(* CODESYS project 18_CS3_EtherCatIOL
   Company: WAGO Contact SA
   Version: 0.0.0.1

Project tree, tasks and I/O mapping:
  Device : 750-8302 PFC300, WAGO, order no. 750-8302, version 6.4.5.11
    application Application
      libraries: Standard, 3.5.18.0 (System)
      task EtherCAT_Task (cyclic, interval t#4ms, priority 1) calls nothing
      task MainTask (cyclic, interval t#50ms, priority 15) calls PLC_PRG
      global variables GVL_IO
      program PLC_PRG [ST]
      program PRG_IOL_Call [ST]
    EtherCAT_Master : EtherCAT Master, CODESYS, version 4.10.0.0
        settings: NetworkName = 'br1'; NetworkName = "br1"; SelectNetworkByName = False; SrcAddress1 = 48; SrcAddress2 = 3731374440
      IOFLD_01_765_1202 : 765-1202/ 16DIO FLD EC 24V 2A, WAGO Kontakttechnik GmbH u. Co. KG, order no. 765-1202, version Revision=16#00000001
          settings: EnableExpertSettings = True; Physical Address of the Slave = 1001; StationAlias = 1001; FixedPhysicalAdress = True; DC sync0 cycletime = 4000; DC enable = 0; DC sync0 enable = 0; DC sync0 factor = 'x 1'; DC sync0 shift time = 0; DC sync1 cycletime = 4000; DC sync1 enable = 0; DC sync1 factor = 'x 1'; DC sync1 shift time = 0; Latch 0 control = 0; Latch 1 control = 0; Number of SDO = 38; Digital Logic Port X02 Pin 4: 0=Digital Input NO normally open,  1=Digital Input NC normally closed, 2=Digital Output, 3=Static On.Value = 2; Digital Logic Port X02 Pin 2: 0=Digital Input NO normally open,  1=Digital Input NC normally closed, 2=Digital Output, 3=Static On.Value = 2; Digital Logic Port X04 Pin 4: 0=Digital Input NO normally open,  1=Digital Input NC normally closed, 2=Digital Output, 3=Static On.Value = 2; Digital Logic Port X04 Pin 2: 0=Digital Input NO normally open,  1=Digital Input NC normally closed, 2=Digital Output, 3=Static On.Value = 2; Digital Logic Port X06 Pin 4: 0=Digital Input NO normally open,  1=Digital Input NC normally closed, 2=Digital Output, 3=Static On.Value = 2; Digital Logic Port X06 Pin 2: 0=Digital Input NO normally open,  1=Digital Input NC normally closed, 2=Digital Output, 3=Static On.Value = 2; Digital Logic Port X08 Pin 4: 0=Digital Input NO normally open,  1=Digital Input NC normally closed, 2=Digital Output, 3=Static On.Value = 2; Digital Logic Port X08 Pin 2: 0=Digital Input NO normally open,  1=Digital Input NC normally closed, 2=Digital Output, 3=Static On.Value = 2
          output Application.GVL_IO.xIOFLD_01_X02_P4_Out : BOOL  // Process Data (Pin2 + Pin4).Bit2
          output Application.GVL_IO.xIOFLD_01_X02_P2_Out : BOOL  // Process Data (Pin2 + Pin4).Bit3
          output Application.GVL_IO.xIOFLD_01_X04_P4_Out : BOOL  // Process Data (Pin2 + Pin4).Bit6
          output Application.GVL_IO.xIOFLD_01_X04_P2_Out : BOOL  // Process Data (Pin2 + Pin4).Bit7
          output Application.GVL_IO.xIOFLD_01_X06_P4_Out : BOOL  // Process Data (Pin2 + Pin4).Bit10
          output Application.GVL_IO.xIOFLD_01_X06_P2_Out : BOOL  // Process Data (Pin2 + Pin4).Bit11
          output Application.GVL_IO.xIOFLD_01_X08_P4_Out : BOOL  // Process Data (Pin2 + Pin4).Bit14
          output Application.GVL_IO.xIOFLD_01_X08_P2_Out : BOOL  // Process Data (Pin2 + Pin4).Bit15
          input  Application.GVL_IO.xIOFLD_01_X01_P4_In : BOOL  // Process Data (Pin2 + Pin4).Bit0
          input  Application.GVL_IO.xIOFLD_01_X01_P2_In : BOOL  // Process Data (Pin2 + Pin4).Bit1
          input  Application.GVL_IO.xIOFLD_01_X03_P4_In : BOOL  // Process Data (Pin2 + Pin4).Bit4
          input  Application.GVL_IO.xIOFLD_01_X03_P2_In : BOOL  // Process Data (Pin2 + Pin4).Bit5
          input  Application.GVL_IO.xIOFLD_01_X05_P4_In : BOOL  // Process Data (Pin2 + Pin4).Bit8
          input  Application.GVL_IO.xIOFLD_01_X05_P2_In : BOOL  // Process Data (Pin2 + Pin4).Bit9
          input  Application.GVL_IO.xIOFLD_01_X07_P4_In : BOOL  // Process Data (Pin2 + Pin4).Bit12
          input  Application.GVL_IO.xIOFLD_01_X07_P2_In : BOOL  // Process Data (Pin2 + Pin4).Bit13
          unmapped channels: Process Data (Pin2 + Pin4), Control Bit, Toggle Bit, ---, ---, ---, ---, ---, ---, Process Data (Pin2 + Pin4), Status Bit, Toggle Bit, ---, ---, ---, ---, ---, ---, New Message Available Flag, ---, ---, ---, ---, ---, ---, ---
      IOFLD_02_765_4201 : 765-4201/ 8P IOLA FLD EC 24V 2A, WAGO Kontakttechnik GmbH u. Co. KG, order no. 765-4201, version Revision=16#00000001
          settings: ModularDevice = True; MDP_InputOffsets = [0,88,0,152,0,168,184,192,448]; MDP_OutputOffsets = [0,16,80,88,104,112,0,128,0]; Physical Address of the Slave = 1002; StationAlias = 1002; FixedPhysicalAdress = True; Sync.Length = 48; Sync.Length = 57; FMMU.Length = 48; FMMU.Length = 57; Number of RxPDOs of the Slave = 7; Number of TxPDOs of the Slave = 9; DC sync0 cycletime = 4000; DC sync1 cycletime = 4000; Number of SDO = 102; Device ID.Index = 16#8000; Device ID.Subindex = 16#04; Device ID.Value = 0; Device ID.Size = 32; Device ID.AbortIfError = FALSE; Device ID.JumpToLine = FALSE; Device ID.Line = 0; Device ID.CompleteAccess = False; Vendor ID.Index = 16#8000; Vendor ID.Subindex = 16#05; Vendor ID.Value = 0; Vendor ID.Size = 32; Vendor ID.AbortIfError = FALSE; Vendor ID.JumpToLine = FALSE; Vendor ID.Line = 0; Vendor ID.CompleteAccess = False; IO-Link Revision 00 = plausibilty check is deactivate, e.g. 11 = V1.1 - plausibilty check is active.Index = 16#8000; IO-Link Revision 00 = plausibilty check is deactivate, e.g. 11 = V1.1 - plausibilty check is active.Subindex = 16#20; IO-Link Revision 00 = plausibilty check is deactivate, e.g. 11 = V1.1 - plausibilty check is active.Value = 0; IO-Link Revision 00 = plausibilty check is deactivate, e.g. 11 = V1.1 - plausibilty check is active.Size = 8; IO-Link Revision 00 = plausibilty check is deactivate, e.g. 11 = V1.1 - plausibilty check is active.AbortIfError = FALSE; IO-Link Revision 00 = plausibilty check is deactivate, e.g. 11 = V1.1 - plausibilty check is active.JumpToLine = FALSE; IO-Link Revision 00 = plausibilty check is deactivate, e.g. 11 = V1.1 - plausibilty check is active.Line = 0; IO-Link Revision 00 = plausibilty check is deactivate, e.g. 11 = V1.1 - plausibilty check is active.CompleteAccess = False; Cycle Time.Index = 16#8000;
            Cycle Time.Subindex = 16#22; Cycle Time.Value = 0; Cycle Time.Size = 8; Cycle Time.AbortIfError = FALSE; Cycle Time.JumpToLine = FALSE; Cycle Time.Line = 0; Cycle Time.CompleteAccess = False; Configured by the plugged slot module, please do not change..Index = 16#8000; Configured by the plugged slot module, please do not change..Subindex = 16#24; Configured by the plugged slot module, please do not change..Value = 135; Configured by the plugged slot module, please do not change..Size = 8; Configured by the plugged slot module, please do not change..AbortIfError = FALSE; Configured by the plugged slot module, please do not change..JumpToLine = FALSE; Configured by the plugged slot module, please do not change..Line = 0; Configured by the plugged slot module, please do not change..CompleteAccess = False; Configured by the plugged slot module, please do not change..Index = 16#8000; Configured by the plugged slot module, please do not change..Subindex = 16#25; Configured by the plugged slot module, please do not change..Value = 135; Configured by the plugged slot module, please do not change..Size = 8; Configured by the plugged slot module, please do not change..AbortIfError = FALSE; Configured by the plugged slot module, please do not change..JumpToLine = FALSE; Configured by the plugged slot module, please do not change..Line = 0; Configured by the plugged slot module, please do not change..CompleteAccess = False; Master Control: 0x0003 = No Data Storage, 0x0023 = Backup + Restore, 0x0043 = Restore.Index = 16#8000; Master Control: 0x0003 = No Data Storage, 0x0023 = Backup + Restore, 0x0043 = Restore.Subindex = 16#28; Master Control: 0x0003 = No Data Storage, 0x0023 = Backup + Restore, 0x0043 = Restore.Value = 3; Master Control: 0x0003 = No Data Storage, 0x0023 = Backup + Restore, 0x0043 = Restore.Size = 16; Master Control: 0x0003 = No Data Storage, 0x0023 = Backup + Restore, 0x0043 = Restore.AbortIfError = FALSE; Master Control: 0x0003 = No Data Storage, 0x0023 = Backup + Restore, 0x0043 = Restore.JumpToLine = FALSE; Master Control: 0x0003 = No Data Storage, 0x0023 = Backup + Restore, 0x0043 = Restore.Line = 0; Master Control: 0x0003 = No Data Storage, 0x0023 = Backup + Restore, 0x0043 = Restore.CompleteAccess = False; Configured by the plugged slot module, please do not change..Index = 16#2100; Configured by the plugged slot module, please do not change..Subindex = 16#24; Configured by the plugged slot module, please do not change..Value = 8; Configured by the plugged slot module, please do not change..Size = 8; Configured by the plugged slot module, please do not change..AbortIfError = FALSE; Configured by the plugged slot module, please do not change..JumpToLine = FALSE; Configured by the plugged slot module, please do not change..Line = 0; Configured by the plugged slot module, please do not change..CompleteAccess = False; Configured by the plugged slot module, please do not change..Index = 16#2100;
            Configured by the plugged slot module, please do not change..Subindex = 16#25; Configured by the plugged slot module, please do not change..Value = 8; Configured by the plugged slot module, please do not change..Size = 8; Configured by the plugged slot module, please do not change..AbortIfError = FALSE; Configured by the plugged slot module, please do not change..JumpToLine = FALSE; Configured by the plugged slot module, please do not change..Line = 0; Configured by the plugged slot module, please do not change..CompleteAccess = False; Configured by the plugged slot module, please do not change..Index = 16#8010; Configured by the plugged slot module, please do not change..Subindex = 16#24; Configured by the plugged slot module, please do not change..Value = 0; Configured by the plugged slot module, please do not change..Size = 8; Configured by the plugged slot module, please do not change..AbortIfError = FALSE; Configured by the plugged slot module, please do not change..JumpToLine = FALSE; Configured by the plugged slot module, please do not change..Line = 0; Configured by the plugged slot module, please do not change..CompleteAccess = False; Configured by the plugged slot module, please do not change..Index = 16#8010; Configured by the plugged slot module, please do not change..Subindex = 16#25; Configured by the plugged slot module, please do not change..Value = 128; Configured by the plugged slot module, please do not change..Size = 8; Configured by the plugged slot module, please do not change..AbortIfError = FALSE; Configured by the plugged slot module, please do not change..JumpToLine = FALSE; Configured by the plugged slot module, please do not change..Line = 0; Configured by the plugged slot module, please do not change..CompleteAccess = False; Configured by the plugged slot module, please do not change..Index = 16#8010; Configured by the plugged slot module, please do not change..Subindex = 16#28; Configured by the plugged slot module, please do not change..Value = 2; Configured by the plugged slot module, please do not change..Size = 16; Configured by the plugged slot module, please do not change..AbortIfError = FALSE; Configured by the plugged slot module, please do not change..JumpToLine = FALSE; Configured by the plugged slot module, please do not change..Line = 0; Configured by the plugged slot module, please do not change..CompleteAccess = False; Configured by the plugged slot module, please do not change..Index = 16#2110; Configured by the plugged slot module, please do not change..Subindex = 16#24; Configured by the plugged slot module, please do not change..Value = 0; Configured by the plugged slot module, please do not change..Size = 8; Configured by the plugged slot module, please do not change..AbortIfError = FALSE; Configured by the plugged slot module, please do not change..JumpToLine = FALSE; Configured by the plugged slot module, please do not change..Line = 0; Configured by the plugged slot module, please do not change..CompleteAccess = False; Configured by the plugged slot module, please do not change..Index = 16#2110;
            Configured by the plugged slot module, please do not change..Subindex = 16#25; Configured by the plugged slot module, please do not change..Value = 0; Configured by the plugged slot module, please do not change..Size = 8; Configured by the plugged slot module, please do not change..AbortIfError = FALSE; Configured by the plugged slot module, please do not change..JumpToLine = FALSE; Configured by the plugged slot module, please do not change..Line = 0; Configured by the plugged slot module, please do not change..CompleteAccess = False; Device ID.Index = 16#8020; Device ID.Subindex = 16#04; Device ID.Value = 0; Device ID.Size = 32; Device ID.AbortIfError = FALSE; Device ID.JumpToLine = FALSE; Device ID.Line = 0; Device ID.CompleteAccess = False; Vendor ID.Index = 16#8020; Vendor ID.Subindex = 16#05; Vendor ID.Value = 0; Vendor ID.Size = 32; Vendor ID.AbortIfError = FALSE; Vendor ID.JumpToLine = FALSE; Vendor ID.Line = 0; Vendor ID.CompleteAccess = False; IO-Link Revision 00 = plausibilty check is deactivate, e.g. 11 = V1.1 - plausibilty check is active.Index = 16#8020; IO-Link Revision 00 = plausibilty check is deactivate, e.g. 11 = V1.1 - plausibilty check is active.Subindex = 16#20; IO-Link Revision 00 = plausibilty check is deactivate, e.g. 11 = V1.1 - plausibilty check is active.Value = 0; IO-Link Revision 00 = plausibilty check is deactivate, e.g. 11 = V1.1 - plausibilty check is active.Size = 8; IO-Link Revision 00 = plausibilty check is deactivate, e.g. 11 = V1.1 - plausibilty check is active.AbortIfError = FALSE; IO-Link Revision 00 = plausibilty check is deactivate, e.g. 11 = V1.1 - plausibilty check is active.JumpToLine = FALSE; IO-Link Revision 00 = plausibilty check is deactivate, e.g. 11 = V1.1 - plausibilty check is active.Line = 0; IO-Link Revision 00 = plausibilty check is deactivate, e.g. 11 = V1.1 - plausibilty check is active.CompleteAccess = False; Cycle Time.Index = 16#8020; Cycle Time.Subindex = 16#22; Cycle Time.Value = 0; Cycle Time.Size = 8; Cycle Time.AbortIfError = FALSE; Cycle Time.JumpToLine = FALSE; Cycle Time.Line = 0; Cycle Time.CompleteAccess = False; Configured by the plugged slot module, please do not change..Index = 16#8020;
            Configured by the plugged slot module, please do not change..Subindex = 16#24; Configured by the plugged slot module, please do not change..Value = 129; Configured by the plugged slot module, please do not change..Size = 8; Configured by the plugged slot module, please do not change..AbortIfError = FALSE; Configured by the plugged slot module, please do not change..JumpToLine = FALSE; Configured by the plugged slot module, please do not change..Line = 0; Configured by the plugged slot module, please do not change..CompleteAccess = False; Configured by the plugged slot module, please do not change..Index = 16#8020; Configured by the plugged slot module, please do not change..Subindex = 16#25; Configured by the plugged slot module, please do not change..Value = 129; Configured by the plugged slot module, please do not change..Size = 8; Configured by the plugged slot module, please do not change..AbortIfError = FALSE; Configured by the plugged slot module, please do not change..JumpToLine = FALSE; Configured by the plugged slot module, please do not change..Line = 0; Configured by the plugged slot module, please do not change..CompleteAccess = False; Master Control: 0x0003 = No Data Storage, 0x0023 = Backup + Restore, 0x0043 = Restore.Index = 16#8020; Master Control: 0x0003 = No Data Storage, 0x0023 = Backup + Restore, 0x0043 = Restore.Subindex = 16#28; Master Control: 0x0003 = No Data Storage, 0x0023 = Backup + Restore, 0x0043 = Restore.Value = 3; Master Control: 0x0003 = No Data Storage, 0x0023 = Backup + Restore, 0x0043 = Restore.Size = 16; Master Control: 0x0003 = No Data Storage, 0x0023 = Backup + Restore, 0x0043 = Restore.AbortIfError = FALSE; Master Control: 0x0003 = No Data Storage, 0x0023 = Backup + Restore, 0x0043 = Restore.JumpToLine = FALSE; Master Control: 0x0003 = No Data Storage, 0x0023 = Backup + Restore, 0x0043 = Restore.Line = 0; Master Control: 0x0003 = No Data Storage, 0x0023 = Backup + Restore, 0x0043 = Restore.CompleteAccess = False; Configured by the plugged slot module, please do not change..Index = 16#2120; Configured by the plugged slot module, please do not change..Subindex = 16#24; Configured by the plugged slot module, please do not change..Value = 2; Configured by the plugged slot module, please do not change..Size = 8; Configured by the plugged slot module, please do not change..AbortIfError = FALSE; Configured by the plugged slot module, please do not change..JumpToLine = FALSE; Configured by the plugged slot module, please do not change..Line = 0; Configured by the plugged slot module, please do not change..CompleteAccess = False; Configured by the plugged slot module, please do not change..Index = 16#2120; Configured by the plugged slot module, please do not change..Subindex = 16#25; Configured by the plugged slot module, please do not change..Value = 2; Configured by the plugged slot module, please do not change..Size = 8; Configured by the plugged slot module, please do not change..AbortIfError = FALSE; Configured by the plugged slot module, please do not change..JumpToLine = FALSE; Configured by the plugged slot module, please do not change..Line = 0; Configured by the plugged slot module, please do not change..CompleteAccess = False; Configured by the plugged slot module, please do not change..Index = 16#8030;
            Configured by the plugged slot module, please do not change..Subindex = 16#24; Configured by the plugged slot module, please do not change..Value = 0; Configured by the plugged slot module, please do not change..Size = 8; Configured by the plugged slot module, please do not change..AbortIfError = FALSE; Configured by the plugged slot module, please do not change..JumpToLine = FALSE; Configured by the plugged slot module, please do not change..Line = 0; Configured by the plugged slot module, please do not change..CompleteAccess = False; Configured by the plugged slot module, please do not change..Index = 16#8030; Configured by the plugged slot module, please do not change..Subindex = 16#25; Configured by the plugged slot module, please do not change..Value = 128; Configured by the plugged slot module, please do not change..Size = 8; Configured by the plugged slot module, please do not change..AbortIfError = FALSE; Configured by the plugged slot module, please do not change..JumpToLine = FALSE; Configured by the plugged slot module, please do not change..Line = 0; Configured by the plugged slot module, please do not change..CompleteAccess = False; Configured by the plugged slot module, please do not change..Index = 16#8030; Configured by the plugged slot module, please do not change..Subindex = 16#28; Configured by the plugged slot module, please do not change..Value = 2; Configured by the plugged slot module, please do not change..Size = 16; Configured by the plugged slot module, please do not change..AbortIfError = FALSE; Configured by the plugged slot module, please do not change..JumpToLine = FALSE; Configured by the plugged slot module, please do not change..Line = 0; Configured by the plugged slot module, please do not change..CompleteAccess = False; Configured by the plugged slot module, please do not change..Index = 16#2130; Configured by the plugged slot module, please do not change..Subindex = 16#24; Configured by the plugged slot module, please do not change..Value = 0; Configured by the plugged slot module, please do not change..Size = 8; Configured by the plugged slot module, please do not change..AbortIfError = FALSE; Configured by the plugged slot module, please do not change..JumpToLine = FALSE; Configured by the plugged slot module, please do not change..Line = 0; Configured by the plugged slot module, please do not change..CompleteAccess = False; Configured by the plugged slot module, please do not change..Index = 16#2130; Configured by the plugged slot module, please do not change..Subindex = 16#25; Configured by the plugged slot module, please do not change..Value = 0; Configured by the plugged slot module, please do not change..Size = 8; Configured by the plugged slot module, please do not change..AbortIfError = FALSE; Configured by the plugged slot module, please do not change..JumpToLine = FALSE; Configured by the plugged slot module, please do not change..Line = 0; Configured by the plugged slot module, please do not change..CompleteAccess = False; Device ID.Index = 16#8040;
            Device ID.Subindex = 16#04; Device ID.Value = 0; Device ID.Size = 32; Device ID.AbortIfError = FALSE; Device ID.JumpToLine = FALSE; Device ID.Line = 0; Device ID.CompleteAccess = False; Vendor ID.Index = 16#8040; Vendor ID.Subindex = 16#05; Vendor ID.Value = 0; Vendor ID.Size = 32; Vendor ID.AbortIfError = FALSE; Vendor ID.JumpToLine = FALSE; Vendor ID.Line = 0; Vendor ID.CompleteAccess = False; IO-Link Revision 00 = plausibilty check is deactivate, e.g. 11 = V1.1 - plausibilty check is active.Index = 16#8040; IO-Link Revision 00 = plausibilty check is deactivate, e.g. 11 = V1.1 - plausibilty check is active.Subindex = 16#20; IO-Link Revision 00 = plausibilty check is deactivate, e.g. 11 = V1.1 - plausibilty check is active.Value = 0; IO-Link Revision 00 = plausibilty check is deactivate, e.g. 11 = V1.1 - plausibilty check is active.Size = 8; IO-Link Revision 00 = plausibilty check is deactivate, e.g. 11 = V1.1 - plausibilty check is active.AbortIfError = FALSE; IO-Link Revision 00 = plausibilty check is deactivate, e.g. 11 = V1.1 - plausibilty check is active.JumpToLine = FALSE; IO-Link Revision 00 = plausibilty check is deactivate, e.g. 11 = V1.1 - plausibilty check is active.Line = 0; IO-Link Revision 00 = plausibilty check is deactivate, e.g. 11 = V1.1 - plausibilty check is active.CompleteAccess = False; Cycle Time.Index = 16#8040; Cycle Time.Subindex = 16#22; Cycle Time.Value = 0; Cycle Time.Size = 8; Cycle Time.AbortIfError = FALSE; Cycle Time.JumpToLine = FALSE; Cycle Time.Line = 0; Cycle Time.CompleteAccess = False; Configured by the plugged slot module, please do not change..Index = 16#8040; Configured by the plugged slot module, please do not change..Subindex = 16#24; Configured by the plugged slot module, please do not change..Value = 129; Configured by the plugged slot module, please do not change..Size = 8; Configured by the plugged slot module, please do not change..AbortIfError = FALSE; Configured by the plugged slot module, please do not change..JumpToLine = FALSE; Configured by the plugged slot module, please do not change..Line = 0; Configured by the plugged slot module, please do not change..CompleteAccess = False; Configured by the plugged slot module, please do not change..Index = 16#8040;
            Configured by the plugged slot module, please do not change..Subindex = 16#25; Configured by the plugged slot module, please do not change..Value = 129; Configured by the plugged slot module, please do not change..Size = 8; Configured by the plugged slot module, please do not change..AbortIfError = FALSE; Configured by the plugged slot module, please do not change..JumpToLine = FALSE; Configured by the plugged slot module, please do not change..Line = 0; Configured by the plugged slot module, please do not change..CompleteAccess = False; Master Control: 0x0003 = No Data Storage, 0x0023 = Backup + Restore, 0x0043 = Restore.Index = 16#8040; Master Control: 0x0003 = No Data Storage, 0x0023 = Backup + Restore, 0x0043 = Restore.Subindex = 16#28; Master Control: 0x0003 = No Data Storage, 0x0023 = Backup + Restore, 0x0043 = Restore.Value = 3; Master Control: 0x0003 = No Data Storage, 0x0023 = Backup + Restore, 0x0043 = Restore.Size = 16; Master Control: 0x0003 = No Data Storage, 0x0023 = Backup + Restore, 0x0043 = Restore.AbortIfError = FALSE; Master Control: 0x0003 = No Data Storage, 0x0023 = Backup + Restore, 0x0043 = Restore.JumpToLine = FALSE; Master Control: 0x0003 = No Data Storage, 0x0023 = Backup + Restore, 0x0043 = Restore.Line = 0; Master Control: 0x0003 = No Data Storage, 0x0023 = Backup + Restore, 0x0043 = Restore.CompleteAccess = False; Configured by the plugged slot module, please do not change..Index = 16#2140; Configured by the plugged slot module, please do not change..Subindex = 16#24; Configured by the plugged slot module, please do not change..Value = 2; Configured by the plugged slot module, please do not change..Size = 8; Configured by the plugged slot module, please do not change..AbortIfError = FALSE; Configured by the plugged slot module, please do not change..JumpToLine = FALSE; Configured by the plugged slot module, please do not change..Line = 0; Configured by the plugged slot module, please do not change..CompleteAccess = False; Configured by the plugged slot module, please do not change..Index = 16#2140; Configured by the plugged slot module, please do not change..Subindex = 16#25; Configured by the plugged slot module, please do not change..Value = 2; Configured by the plugged slot module, please do not change..Size = 8; Configured by the plugged slot module, please do not change..AbortIfError = FALSE; Configured by the plugged slot module, please do not change..JumpToLine = FALSE; Configured by the plugged slot module, please do not change..Line = 0; Configured by the plugged slot module, please do not change..CompleteAccess = False; Configured by the plugged slot module, please do not change..Index = 16#8050; Configured by the plugged slot module, please do not change..Subindex = 16#24; Configured by the plugged slot module, please do not change..Value = 128; Configured by the plugged slot module, please do not change..Size = 8; Configured by the plugged slot module, please do not change..AbortIfError = FALSE; Configured by the plugged slot module, please do not change..JumpToLine = FALSE; Configured by the plugged slot module, please do not change..Line = 0; Configured by the plugged slot module, please do not change..CompleteAccess = False; Configured by the plugged slot module, please do not change..Index = 16#8050;
            Configured by the plugged slot module, please do not change..Subindex = 16#25; Configured by the plugged slot module, please do not change..Value = 0; Configured by the plugged slot module, please do not change..Size = 8; Configured by the plugged slot module, please do not change..AbortIfError = FALSE; Configured by the plugged slot module, please do not change..JumpToLine = FALSE; Configured by the plugged slot module, please do not change..Line = 0; Configured by the plugged slot module, please do not change..CompleteAccess = False; Configured by the plugged slot module, please do not change..Index = 16#8050; Configured by the plugged slot module, please do not change..Subindex = 16#28; Configured by the plugged slot module, please do not change..Value = 1; Configured by the plugged slot module, please do not change..Size = 16; Configured by the plugged slot module, please do not change..AbortIfError = FALSE; Configured by the plugged slot module, please do not change..JumpToLine = FALSE; Configured by the plugged slot module, please do not change..Line = 0; Configured by the plugged slot module, please do not change..CompleteAccess = False; Configured by the plugged slot module, please do not change..Index = 16#2150; Configured by the plugged slot module, please do not change..Subindex = 16#24; Configured by the plugged slot module, please do not change..Value = 0; Configured by the plugged slot module, please do not change..Size = 8; Configured by the plugged slot module, please do not change..AbortIfError = FALSE; Configured by the plugged slot module, please do not change..JumpToLine = FALSE; Configured by the plugged slot module, please do not change..Line = 0; Configured by the plugged slot module, please do not change..CompleteAccess = False; Configured by the plugged slot module, please do not change..Index = 16#2150; Configured by the plugged slot module, please do not change..Subindex = 16#25; Configured by the plugged slot module, please do not change..Value = 0; Configured by the plugged slot module, please do not change..Size = 8; Configured by the plugged slot module, please do not change..AbortIfError = FALSE; Configured by the plugged slot module, please do not change..JumpToLine = FALSE; Configured by the plugged slot module, please do not change..Line = 0; Configured by the plugged slot module, please do not change..CompleteAccess = False; Device ID.Index = 16#8060; Device ID.Subindex = 16#04; Device ID.Value = 0; Device ID.Size = 32; Device ID.AbortIfError = FALSE; Device ID.JumpToLine = FALSE; Device ID.Line = 0; Device ID.CompleteAccess = False; Vendor ID.Index = 16#8060;
            Vendor ID.Subindex = 16#05; Vendor ID.Value = 0; Vendor ID.Size = 32; Vendor ID.AbortIfError = FALSE; Vendor ID.JumpToLine = FALSE; Vendor ID.Line = 0; Vendor ID.CompleteAccess = False; IO-Link Revision 00 = plausibilty check is deactivate, e.g. 11 = V1.1 - plausibilty check is active.Index = 16#8060; IO-Link Revision 00 = plausibilty check is deactivate, e.g. 11 = V1.1 - plausibilty check is active.Subindex = 16#20; IO-Link Revision 00 = plausibilty check is deactivate, e.g. 11 = V1.1 - plausibilty check is active.Value = 0; IO-Link Revision 00 = plausibilty check is deactivate, e.g. 11 = V1.1 - plausibilty check is active.Size = 8; IO-Link Revision 00 = plausibilty check is deactivate, e.g. 11 = V1.1 - plausibilty check is active.AbortIfError = FALSE; IO-Link Revision 00 = plausibilty check is deactivate, e.g. 11 = V1.1 - plausibilty check is active.JumpToLine = FALSE; IO-Link Revision 00 = plausibilty check is deactivate, e.g. 11 = V1.1 - plausibilty check is active.Line = 0; IO-Link Revision 00 = plausibilty check is deactivate, e.g. 11 = V1.1 - plausibilty check is active.CompleteAccess = False; Cycle Time.Index = 16#8060; Cycle Time.Subindex = 16#22; Cycle Time.Value = 0; Cycle Time.Size = 8; Cycle Time.AbortIfError = FALSE; Cycle Time.JumpToLine = FALSE; Cycle Time.Line = 0; Cycle Time.CompleteAccess = False; Configured by the plugged slot module, please do not change..Index = 16#8060; Configured by the plugged slot module, please do not change..Subindex = 16#24; Configured by the plugged slot module, please do not change..Value = 159; Configured by the plugged slot module, please do not change..Size = 8; Configured by the plugged slot module, please do not change..AbortIfError = FALSE; Configured by the plugged slot module, please do not change..JumpToLine = FALSE; Configured by the plugged slot module, please do not change..Line = 0; Configured by the plugged slot module, please do not change..CompleteAccess = False; Configured by the plugged slot module, please do not change..Index = 16#8060; Configured by the plugged slot module, please do not change..Subindex = 16#25; Configured by the plugged slot module, please do not change..Value = 159; Configured by the plugged slot module, please do not change..Size = 8; Configured by the plugged slot module, please do not change..AbortIfError = FALSE; Configured by the plugged slot module, please do not change..JumpToLine = FALSE; Configured by the plugged slot module, please do not change..Line = 0; Configured by the plugged slot module, please do not change..CompleteAccess = False; Master Control: 0x0003 = No Data Storage, 0x0023 = Backup + Restore, 0x0043 = Restore.Index = 16#8060;
            Master Control: 0x0003 = No Data Storage, 0x0023 = Backup + Restore, 0x0043 = Restore.Subindex = 16#28; Master Control: 0x0003 = No Data Storage, 0x0023 = Backup + Restore, 0x0043 = Restore.Value = 3; Master Control: 0x0003 = No Data Storage, 0x0023 = Backup + Restore, 0x0043 = Restore.Size = 16; Master Control: 0x0003 = No Data Storage, 0x0023 = Backup + Restore, 0x0043 = Restore.AbortIfError = FALSE; Master Control: 0x0003 = No Data Storage, 0x0023 = Backup + Restore, 0x0043 = Restore.JumpToLine = FALSE; Master Control: 0x0003 = No Data Storage, 0x0023 = Backup + Restore, 0x0043 = Restore.Line = 0; Master Control: 0x0003 = No Data Storage, 0x0023 = Backup + Restore, 0x0043 = Restore.CompleteAccess = False; Configured by the plugged slot module, please do not change..Index = 16#2160; Configured by the plugged slot module, please do not change..Subindex = 16#24; Configured by the plugged slot module, please do not change..Value = 32; Configured by the plugged slot module, please do not change..Size = 8; Configured by the plugged slot module, please do not change..AbortIfError = FALSE; Configured by the plugged slot module, please do not change..JumpToLine = FALSE; Configured by the plugged slot module, please do not change..Line = 0; Configured by the plugged slot module, please do not change..CompleteAccess = False; Configured by the plugged slot module, please do not change..Index = 16#2160; Configured by the plugged slot module, please do not change..Subindex = 16#25; Configured by the plugged slot module, please do not change..Value = 32; Configured by the plugged slot module, please do not change..Size = 8; Configured by the plugged slot module, please do not change..AbortIfError = FALSE; Configured by the plugged slot module, please do not change..JumpToLine = FALSE; Configured by the plugged slot module, please do not change..Line = 0; Configured by the plugged slot module, please do not change..CompleteAccess = False; Configured by the plugged slot module, please do not change..Index = 16#8070; Configured by the plugged slot module, please do not change..Subindex = 16#24; Configured by the plugged slot module, please do not change..Value = 128; Configured by the plugged slot module, please do not change..Size = 8; Configured by the plugged slot module, please do not change..AbortIfError = FALSE; Configured by the plugged slot module, please do not change..JumpToLine = FALSE; Configured by the plugged slot module, please do not change..Line = 0; Configured by the plugged slot module, please do not change..CompleteAccess = False; Configured by the plugged slot module, please do not change..Index = 16#8070; Configured by the plugged slot module, please do not change..Subindex = 16#25; Configured by the plugged slot module, please do not change..Value = 0; Configured by the plugged slot module, please do not change..Size = 8; Configured by the plugged slot module, please do not change..AbortIfError = FALSE; Configured by the plugged slot module, please do not change..JumpToLine = FALSE; Configured by the plugged slot module, please do not change..Line = 0; Configured by the plugged slot module, please do not change..CompleteAccess = False; Configured by the plugged slot module, please do not change..Index = 16#8070;
            Configured by the plugged slot module, please do not change..Subindex = 16#28; Configured by the plugged slot module, please do not change..Value = 1; Configured by the plugged slot module, please do not change..Size = 16; Configured by the plugged slot module, please do not change..AbortIfError = FALSE; Configured by the plugged slot module, please do not change..JumpToLine = FALSE; Configured by the plugged slot module, please do not change..Line = 0; Configured by the plugged slot module, please do not change..CompleteAccess = False; Configured by the plugged slot module, please do not change..Index = 16#2170; Configured by the plugged slot module, please do not change..Subindex = 16#24; Configured by the plugged slot module, please do not change..Value = 0; Configured by the plugged slot module, please do not change..Size = 8; Configured by the plugged slot module, please do not change..AbortIfError = FALSE; Configured by the plugged slot module, please do not change..JumpToLine = FALSE; Configured by the plugged slot module, please do not change..Line = 0; Configured by the plugged slot module, please do not change..CompleteAccess = False; Configured by the plugged slot module, please do not change..Index = 16#2170; Configured by the plugged slot module, please do not change..Subindex = 16#25; Configured by the plugged slot module, please do not change..Value = 0; Configured by the plugged slot module, please do not change..Size = 8; Configured by the plugged slot module, please do not change..AbortIfError = FALSE; Configured by the plugged slot module, please do not change..JumpToLine = FALSE; Configured by the plugged slot module, please do not change..Line = 0; Configured by the plugged slot module, please do not change..CompleteAccess = False; Force Mode Setting: 0=Force mode enable, 1=Force mode disable.Index = 16#2000; Force Mode Setting: 0=Force mode enable, 1=Force mode disable.Subindex = 16#00; Force Mode Setting: 0=Force mode enable, 1=Force mode disable.Value = 0; Force Mode Setting: 0=Force mode enable, 1=Force mode disable.Size = 8; Force Mode Setting: 0=Force mode enable, 1=Force mode disable.AbortIfError = FALSE; Force Mode Setting: 0=Force mode enable, 1=Force mode disable.JumpToLine = FALSE; Force Mode Setting: 0=Force mode enable, 1=Force mode disable.Line = 0; Force Mode Setting: 0=Force mode enable, 1=Force mode disable.CompleteAccess = False; PD-Layout Configuration: 0=Port Based, 1=Pin Based.Index = 16#2001; PD-Layout Configuration: 0=Port Based, 1=Pin Based.Subindex = 16#00; PD-Layout Configuration: 0=Port Based, 1=Pin Based.Value = 0; PD-Layout Configuration: 0=Port Based, 1=Pin Based.Size = 8; PD-Layout Configuration: 0=Port Based, 1=Pin Based.AbortIfError = FALSE; PD-Layout Configuration: 0=Port Based, 1=Pin Based.JumpToLine = FALSE; PD-Layout Configuration: 0=Port Based, 1=Pin Based.Line = 0; PD-Layout Configuration: 0=Port Based, 1=Pin Based.CompleteAccess = False; DO Substitute Mode: 0=Set Low, 1=Substitute Value, 2=Hold last.Index = 16#2002;
            DO Substitute Mode: 0=Set Low, 1=Substitute Value, 2=Hold last.Subindex = 16#01; DO Substitute Mode: 0=Set Low, 1=Substitute Value, 2=Hold last.Value = 0; DO Substitute Mode: 0=Set Low, 1=Substitute Value, 2=Hold last.Size = 8; DO Substitute Mode: 0=Set Low, 1=Substitute Value, 2=Hold last.AbortIfError = FALSE; DO Substitute Mode: 0=Set Low, 1=Substitute Value, 2=Hold last.JumpToLine = FALSE; DO Substitute Mode: 0=Set Low, 1=Substitute Value, 2=Hold last.Line = 0; DO Substitute Mode: 0=Set Low, 1=Substitute Value, 2=Hold last.CompleteAccess = False; DO Substitute Value.Index = 16#2002; DO Substitute Value.Subindex = 16#02; DO Substitute Value.Value = 0; DO Substitute Value.Size = 16; DO Substitute Value.AbortIfError = FALSE; DO Substitute Value.JumpToLine = FALSE; DO Substitute Value.Line = 0; DO Substitute Value.CompleteAccess = False; Disable BT: 0=activation of BT interface is allowed, 1=disable activation of BT interface.Index = 16#2003; Disable BT: 0=activation of BT interface is allowed, 1=disable activation of BT interface.Subindex = 16#01; Disable BT: 0=activation of BT interface is allowed, 1=disable activation of BT interface.Value = 0; Disable BT: 0=activation of BT interface is allowed, 1=disable activation of BT interface.Size = 8; Disable BT: 0=activation of BT interface is allowed, 1=disable activation of BT interface.AbortIfError = FALSE; Disable BT: 0=activation of BT interface is allowed, 1=disable activation of BT interface.JumpToLine = FALSE; Disable BT: 0=activation of BT interface is allowed, 1=disable activation of BT interface.Line = 0; Disable BT: 0=activation of BT interface is allowed, 1=disable activation of BT interface.CompleteAccess = False; BT Timeout: Time out to monitor the BT connection in seconds, input range 6..59s.Index = 16#2003; BT Timeout: Time out to monitor the BT connection in seconds, input range 6..59s.Subindex = 16#02; BT Timeout: Time out to monitor the BT connection in seconds, input range 6..59s.Value = 30; BT Timeout: Time out to monitor the BT connection in seconds, input range 6..59s.Size = 16; BT Timeout: Time out to monitor the BT connection in seconds, input range 6..59s.AbortIfError = FALSE; BT Timeout: Time out to monitor the BT connection in seconds, input range 6..59s.JumpToLine = FALSE; BT Timeout: Time out to monitor the BT connection in seconds, input range 6..59s.Line = 0; BT Timeout: Time out to monitor the BT connection in seconds, input range 6..59s.CompleteAccess = False; Port X01 Pin CQ - DI Invert: false=Digital Input NO normally open,  true=Digital Input NC normally closed.Index = 16#2100; Port X01 Pin CQ - DI Invert: false=Digital Input NO normally open,  true=Digital Input NC normally closed.Subindex = 16#01; Port X01 Pin CQ - DI Invert: false=Digital Input NO normally open,  true=Digital Input NC normally closed.Value = 0; Port X01 Pin CQ - DI Invert: false=Digital Input NO normally open,  true=Digital Input NC normally closed.Size = 8; Port X01 Pin CQ - DI Invert: false=Digital Input NO normally open,  true=Digital Input NC normally closed.AbortIfError = FALSE; Port X01 Pin CQ - DI Invert: false=Digital Input NO normally open,  true=Digital Input NC normally closed.JumpToLine = FALSE; Port X01 Pin CQ - DI Invert: false=Digital Input NO normally open,  true=Digital Input NC normally closed.Line = 0; Port X01 Pin CQ - DI Invert: false=Digital Input NO normally open,  true=Digital Input NC normally closed.CompleteAccess = False; Port X01 Pin CQ - DI Filter Time: 0=no Filter, 30=3ms, 150=15ms, 200=20ms.Index = 16#2100;
            Port X01 Pin CQ - DI Filter Time: 0=no Filter, 30=3ms, 150=15ms, 200=20ms.Subindex = 16#02; Port X01 Pin CQ - DI Filter Time: 0=no Filter, 30=3ms, 150=15ms, 200=20ms.Value = 0; Port X01 Pin CQ - DI Filter Time: 0=no Filter, 30=3ms, 150=15ms, 200=20ms.Size = 8; Port X01 Pin CQ - DI Filter Time: 0=no Filter, 30=3ms, 150=15ms, 200=20ms.AbortIfError = FALSE; Port X01 Pin CQ - DI Filter Time: 0=no Filter, 30=3ms, 150=15ms, 200=20ms.JumpToLine = FALSE; Port X01 Pin CQ - DI Filter Time: 0=no Filter, 30=3ms, 150=15ms, 200=20ms.Line = 0; Port X01 Pin CQ - DI Filter Time: 0=no Filter, 30=3ms, 150=15ms, 200=20ms.CompleteAccess = False; Port X01 Pin CQ - DO Static On: false=off, true=on.Index = 16#2100; Port X01 Pin CQ - DO Static On: false=off, true=on.Subindex = 16#03; Port X01 Pin CQ - DO Static On: false=off, true=on.Value = 0; Port X01 Pin CQ - DO Static On: false=off, true=on.Size = 8; Port X01 Pin CQ - DO Static On: false=off, true=on.AbortIfError = FALSE; Port X01 Pin CQ - DO Static On: false=off, true=on.JumpToLine = FALSE; Port X01 Pin CQ - DO Static On: false=off, true=on.Line = 0; Port X01 Pin CQ - DO Static On: false=off, true=on.CompleteAccess = False; Port X01 Pin IQ - Digital Mode: 0=Digital Input NO normally open,  1=Digital Input NC normally closed, 2=Digital Output, 3=Static On, 4=Not supported.Index = 16#2100; Port X01 Pin IQ - Digital Mode: 0=Digital Input NO normally open,  1=Digital Input NC normally closed, 2=Digital Output, 3=Static On, 4=Not supported.Subindex = 16#04; Port X01 Pin IQ - Digital Mode: 0=Digital Input NO normally open,  1=Digital Input NC normally closed, 2=Digital Output, 3=Static On, 4=Not supported.Value = 4; Port X01 Pin IQ - Digital Mode: 0=Digital Input NO normally open,  1=Digital Input NC normally closed, 2=Digital Output, 3=Static On, 4=Not supported.Size = 8; Port X01 Pin IQ - Digital Mode: 0=Digital Input NO normally open,  1=Digital Input NC normally closed, 2=Digital Output, 3=Static On, 4=Not supported.AbortIfError = FALSE; Port X01 Pin IQ - Digital Mode: 0=Digital Input NO normally open,  1=Digital Input NC normally closed, 2=Digital Output, 3=Static On, 4=Not supported.JumpToLine = FALSE; Port X01 Pin IQ - Digital Mode: 0=Digital Input NO normally open,  1=Digital Input NC normally closed, 2=Digital Output, 3=Static On, 4=Not supported.Line = 0; Port X01 Pin IQ - Digital Mode: 0=Digital Input NO normally open,  1=Digital Input NC normally closed, 2=Digital Output, 3=Static On, 4=Not supported.CompleteAccess = False; Port X01 Pin IQ - DI Filter Time: 0=no Filter, 30=3ms, 150=15ms, 200=20ms.Index = 16#2100; Port X01 Pin IQ - DI Filter Time: 0=no Filter, 30=3ms, 150=15ms, 200=20ms.Subindex = 16#05; Port X01 Pin IQ - DI Filter Time: 0=no Filter, 30=3ms, 150=15ms, 200=20ms.Value = 0; Port X01 Pin IQ - DI Filter Time: 0=no Filter, 30=3ms, 150=15ms, 200=20ms.Size = 8; Port X01 Pin IQ - DI Filter Time: 0=no Filter, 30=3ms, 150=15ms, 200=20ms.AbortIfError = FALSE; Port X01 Pin IQ - DI Filter Time: 0=no Filter, 30=3ms, 150=15ms, 200=20ms.JumpToLine = FALSE; Port X01 Pin IQ - DI Filter Time: 0=no Filter, 30=3ms, 150=15ms, 200=20ms.Line = 0; Port X01 Pin IQ - DI Filter Time: 0=no Filter, 30=3ms, 150=15ms, 200=20ms.CompleteAccess = False; Port X02 Pin CQ - DI Invert: false=Digital Input NO normally open,  true=Digital Input NC normally closed.Index = 16#2110; Port X02 Pin CQ - DI Invert: false=Digital Input NO normally open,  true=Digital Input NC normally closed.Subindex = 16#01; Port X02 Pin CQ - DI Invert: false=Digital Input NO normally open,  true=Digital Input NC normally closed.Value = 0; Port X02 Pin CQ - DI Invert: false=Digital Input NO normally open,  true=Digital Input NC normally closed.Size = 8; Port X02 Pin CQ - DI Invert: false=Digital Input NO normally open,  true=Digital Input NC normally closed.AbortIfError = FALSE; Port X02 Pin CQ - DI Invert: false=Digital Input NO normally open,  true=Digital Input NC normally closed.JumpToLine = FALSE; Port X02 Pin CQ - DI Invert: false=Digital Input NO normally open,  true=Digital Input NC normally closed.Line = 0; Port X02 Pin CQ - DI Invert: false=Digital Input NO normally open,  true=Digital Input NC normally closed.CompleteAccess = False; Port X02 Pin CQ - DI Filter Time: 0=no Filter, 30=3ms, 150=15ms, 200=20ms.Index = 16#2110;
            Port X02 Pin CQ - DI Filter Time: 0=no Filter, 30=3ms, 150=15ms, 200=20ms.Subindex = 16#02; Port X02 Pin CQ - DI Filter Time: 0=no Filter, 30=3ms, 150=15ms, 200=20ms.Value = 0; Port X02 Pin CQ - DI Filter Time: 0=no Filter, 30=3ms, 150=15ms, 200=20ms.Size = 8; Port X02 Pin CQ - DI Filter Time: 0=no Filter, 30=3ms, 150=15ms, 200=20ms.AbortIfError = FALSE; Port X02 Pin CQ - DI Filter Time: 0=no Filter, 30=3ms, 150=15ms, 200=20ms.JumpToLine = FALSE; Port X02 Pin CQ - DI Filter Time: 0=no Filter, 30=3ms, 150=15ms, 200=20ms.Line = 0; Port X02 Pin CQ - DI Filter Time: 0=no Filter, 30=3ms, 150=15ms, 200=20ms.CompleteAccess = False; Port X02 Pin CQ - DO Static On: false=off, true=on.Index = 16#2110; Port X02 Pin CQ - DO Static On: false=off, true=on.Subindex = 16#03; Port X02 Pin CQ - DO Static On: false=off, true=on.Value = 0; Port X02 Pin CQ - DO Static On: false=off, true=on.Size = 8; Port X02 Pin CQ - DO Static On: false=off, true=on.AbortIfError = FALSE; Port X02 Pin CQ - DO Static On: false=off, true=on.JumpToLine = FALSE; Port X02 Pin CQ - DO Static On: false=off, true=on.Line = 0; Port X02 Pin CQ - DO Static On: false=off, true=on.CompleteAccess = False; Port X02 Pin IQ - Digital Mode: 0=Digital Input NO normally open,  1=Digital Input NC normally closed, 2=Digital Output, 3=Static On, 4=Not supported.Index = 16#2110; Port X02 Pin IQ - Digital Mode: 0=Digital Input NO normally open,  1=Digital Input NC normally closed, 2=Digital Output, 3=Static On, 4=Not supported.Subindex = 16#04; Port X02 Pin IQ - Digital Mode: 0=Digital Input NO normally open,  1=Digital Input NC normally closed, 2=Digital Output, 3=Static On, 4=Not supported.Value = 4; Port X02 Pin IQ - Digital Mode: 0=Digital Input NO normally open,  1=Digital Input NC normally closed, 2=Digital Output, 3=Static On, 4=Not supported.Size = 8; Port X02 Pin IQ - Digital Mode: 0=Digital Input NO normally open,  1=Digital Input NC normally closed, 2=Digital Output, 3=Static On, 4=Not supported.AbortIfError = FALSE; Port X02 Pin IQ - Digital Mode: 0=Digital Input NO normally open,  1=Digital Input NC normally closed, 2=Digital Output, 3=Static On, 4=Not supported.JumpToLine = FALSE; Port X02 Pin IQ - Digital Mode: 0=Digital Input NO normally open,  1=Digital Input NC normally closed, 2=Digital Output, 3=Static On, 4=Not supported.Line = 0; Port X02 Pin IQ - Digital Mode: 0=Digital Input NO normally open,  1=Digital Input NC normally closed, 2=Digital Output, 3=Static On, 4=Not supported.CompleteAccess = False; Port X02 Pin IQ - DI Filter Time: 0=no Filter, 30=3ms, 150=15ms, 200=20ms.Index = 16#2110; Port X02 Pin IQ - DI Filter Time: 0=no Filter, 30=3ms, 150=15ms, 200=20ms.Subindex = 16#05; Port X02 Pin IQ - DI Filter Time: 0=no Filter, 30=3ms, 150=15ms, 200=20ms.Value = 0; Port X02 Pin IQ - DI Filter Time: 0=no Filter, 30=3ms, 150=15ms, 200=20ms.Size = 8; Port X02 Pin IQ - DI Filter Time: 0=no Filter, 30=3ms, 150=15ms, 200=20ms.AbortIfError = FALSE; Port X02 Pin IQ - DI Filter Time: 0=no Filter, 30=3ms, 150=15ms, 200=20ms.JumpToLine = FALSE; Port X02 Pin IQ - DI Filter Time: 0=no Filter, 30=3ms, 150=15ms, 200=20ms.Line = 0; Port X02 Pin IQ - DI Filter Time: 0=no Filter, 30=3ms, 150=15ms, 200=20ms.CompleteAccess = False; Port X03 Pin CQ - DI Invert: false=Digital Input NO normally open,  true=Digital Input NC normally closed.Index = 16#2120; Port X03 Pin CQ - DI Invert: false=Digital Input NO normally open,  true=Digital Input NC normally closed.Subindex = 16#01; Port X03 Pin CQ - DI Invert: false=Digital Input NO normally open,  true=Digital Input NC normally closed.Value = 0; Port X03 Pin CQ - DI Invert: false=Digital Input NO normally open,  true=Digital Input NC normally closed.Size = 8; Port X03 Pin CQ - DI Invert: false=Digital Input NO normally open,  true=Digital Input NC normally closed.AbortIfError = FALSE; Port X03 Pin CQ - DI Invert: false=Digital Input NO normally open,  true=Digital Input NC normally closed.JumpToLine = FALSE; Port X03 Pin CQ - DI Invert: false=Digital Input NO normally open,  true=Digital Input NC normally closed.Line = 0; Port X03 Pin CQ - DI Invert: false=Digital Input NO normally open,  true=Digital Input NC normally closed.CompleteAccess = False; Port X03 Pin CQ - DI Filter Time: 0=no Filter, 30=3ms, 150=15ms, 200=20ms.Index = 16#2120;
            Port X03 Pin CQ - DI Filter Time: 0=no Filter, 30=3ms, 150=15ms, 200=20ms.Subindex = 16#02; Port X03 Pin CQ - DI Filter Time: 0=no Filter, 30=3ms, 150=15ms, 200=20ms.Value = 0; Port X03 Pin CQ - DI Filter Time: 0=no Filter, 30=3ms, 150=15ms, 200=20ms.Size = 8; Port X03 Pin CQ - DI Filter Time: 0=no Filter, 30=3ms, 150=15ms, 200=20ms.AbortIfError = FALSE; Port X03 Pin CQ - DI Filter Time: 0=no Filter, 30=3ms, 150=15ms, 200=20ms.JumpToLine = FALSE; Port X03 Pin CQ - DI Filter Time: 0=no Filter, 30=3ms, 150=15ms, 200=20ms.Line = 0; Port X03 Pin CQ - DI Filter Time: 0=no Filter, 30=3ms, 150=15ms, 200=20ms.CompleteAccess = False; Port X03 Pin CQ - DO Static On: false=off, true=on.Index = 16#2120; Port X03 Pin CQ - DO Static On: false=off, true=on.Subindex = 16#03; Port X03 Pin CQ - DO Static On: false=off, true=on.Value = 0; Port X03 Pin CQ - DO Static On: false=off, true=on.Size = 8; Port X03 Pin CQ - DO Static On: false=off, true=on.AbortIfError = FALSE; Port X03 Pin CQ - DO Static On: false=off, true=on.JumpToLine = FALSE; Port X03 Pin CQ - DO Static On: false=off, true=on.Line = 0; Port X03 Pin CQ - DO Static On: false=off, true=on.CompleteAccess = False; Port X03 Pin IQ - Digital Mode: 0=Digital Input NO normally open,  1=Digital Input NC normally closed, 2=Digital Output, 3=Static On, 4=Not supported.Index = 16#2120; Port X03 Pin IQ - Digital Mode: 0=Digital Input NO normally open,  1=Digital Input NC normally closed, 2=Digital Output, 3=Static On, 4=Not supported.Subindex = 16#04; Port X03 Pin IQ - Digital Mode: 0=Digital Input NO normally open,  1=Digital Input NC normally closed, 2=Digital Output, 3=Static On, 4=Not supported.Value = 4; Port X03 Pin IQ - Digital Mode: 0=Digital Input NO normally open,  1=Digital Input NC normally closed, 2=Digital Output, 3=Static On, 4=Not supported.Size = 8; Port X03 Pin IQ - Digital Mode: 0=Digital Input NO normally open,  1=Digital Input NC normally closed, 2=Digital Output, 3=Static On, 4=Not supported.AbortIfError = FALSE; Port X03 Pin IQ - Digital Mode: 0=Digital Input NO normally open,  1=Digital Input NC normally closed, 2=Digital Output, 3=Static On, 4=Not supported.JumpToLine = FALSE; Port X03 Pin IQ - Digital Mode: 0=Digital Input NO normally open,  1=Digital Input NC normally closed, 2=Digital Output, 3=Static On, 4=Not supported.Line = 0; Port X03 Pin IQ - Digital Mode: 0=Digital Input NO normally open,  1=Digital Input NC normally closed, 2=Digital Output, 3=Static On, 4=Not supported.CompleteAccess = False; Port X03 Pin IQ - DI Filter Time: 0=no Filter, 30=3ms, 150=15ms, 200=20ms.Index = 16#2120; Port X03 Pin IQ - DI Filter Time: 0=no Filter, 30=3ms, 150=15ms, 200=20ms.Subindex = 16#05; Port X03 Pin IQ - DI Filter Time: 0=no Filter, 30=3ms, 150=15ms, 200=20ms.Value = 0; Port X03 Pin IQ - DI Filter Time: 0=no Filter, 30=3ms, 150=15ms, 200=20ms.Size = 8; Port X03 Pin IQ - DI Filter Time: 0=no Filter, 30=3ms, 150=15ms, 200=20ms.AbortIfError = FALSE; Port X03 Pin IQ - DI Filter Time: 0=no Filter, 30=3ms, 150=15ms, 200=20ms.JumpToLine = FALSE; Port X03 Pin IQ - DI Filter Time: 0=no Filter, 30=3ms, 150=15ms, 200=20ms.Line = 0; Port X03 Pin IQ - DI Filter Time: 0=no Filter, 30=3ms, 150=15ms, 200=20ms.CompleteAccess = False; Port X04 Pin CQ - DI Invert: false=Digital Input NO normally open,  true=Digital Input NC normally closed.Index = 16#2130; Port X04 Pin CQ - DI Invert: false=Digital Input NO normally open,  true=Digital Input NC normally closed.Subindex = 16#01; Port X04 Pin CQ - DI Invert: false=Digital Input NO normally open,  true=Digital Input NC normally closed.Value = 0; Port X04 Pin CQ - DI Invert: false=Digital Input NO normally open,  true=Digital Input NC normally closed.Size = 8; Port X04 Pin CQ - DI Invert: false=Digital Input NO normally open,  true=Digital Input NC normally closed.AbortIfError = FALSE; Port X04 Pin CQ - DI Invert: false=Digital Input NO normally open,  true=Digital Input NC normally closed.JumpToLine = FALSE; Port X04 Pin CQ - DI Invert: false=Digital Input NO normally open,  true=Digital Input NC normally closed.Line = 0; Port X04 Pin CQ - DI Invert: false=Digital Input NO normally open,  true=Digital Input NC normally closed.CompleteAccess = False; Port X04 Pin CQ - DI Filter Time: 0=no Filter, 30=3ms, 150=15ms, 200=20ms.Index = 16#2130;
            Port X04 Pin CQ - DI Filter Time: 0=no Filter, 30=3ms, 150=15ms, 200=20ms.Subindex = 16#02; Port X04 Pin CQ - DI Filter Time: 0=no Filter, 30=3ms, 150=15ms, 200=20ms.Value = 0; Port X04 Pin CQ - DI Filter Time: 0=no Filter, 30=3ms, 150=15ms, 200=20ms.Size = 8; Port X04 Pin CQ - DI Filter Time: 0=no Filter, 30=3ms, 150=15ms, 200=20ms.AbortIfError = FALSE; Port X04 Pin CQ - DI Filter Time: 0=no Filter, 30=3ms, 150=15ms, 200=20ms.JumpToLine = FALSE; Port X04 Pin CQ - DI Filter Time: 0=no Filter, 30=3ms, 150=15ms, 200=20ms.Line = 0; Port X04 Pin CQ - DI Filter Time: 0=no Filter, 30=3ms, 150=15ms, 200=20ms.CompleteAccess = False; Port X04 Pin CQ - DO Static On: false=off, true=on.Index = 16#2130; Port X04 Pin CQ - DO Static On: false=off, true=on.Subindex = 16#03; Port X04 Pin CQ - DO Static On: false=off, true=on.Value = 0; Port X04 Pin CQ - DO Static On: false=off, true=on.Size = 8; Port X04 Pin CQ - DO Static On: false=off, true=on.AbortIfError = FALSE; Port X04 Pin CQ - DO Static On: false=off, true=on.JumpToLine = FALSE; Port X04 Pin CQ - DO Static On: false=off, true=on.Line = 0; Port X04 Pin CQ - DO Static On: false=off, true=on.CompleteAccess = False; Port X04 Pin IQ - Digital Mode: 0=Digital Input NO normally open,  1=Digital Input NC normally closed, 2=Digital Output, 3=Static On, 4=Not supported.Index = 16#2130; Port X04 Pin IQ - Digital Mode: 0=Digital Input NO normally open,  1=Digital Input NC normally closed, 2=Digital Output, 3=Static On, 4=Not supported.Subindex = 16#04; Port X04 Pin IQ - Digital Mode: 0=Digital Input NO normally open,  1=Digital Input NC normally closed, 2=Digital Output, 3=Static On, 4=Not supported.Value = 4; Port X04 Pin IQ - Digital Mode: 0=Digital Input NO normally open,  1=Digital Input NC normally closed, 2=Digital Output, 3=Static On, 4=Not supported.Size = 8; Port X04 Pin IQ - Digital Mode: 0=Digital Input NO normally open,  1=Digital Input NC normally closed, 2=Digital Output, 3=Static On, 4=Not supported.AbortIfError = FALSE; Port X04 Pin IQ - Digital Mode: 0=Digital Input NO normally open,  1=Digital Input NC normally closed, 2=Digital Output, 3=Static On, 4=Not supported.JumpToLine = FALSE; Port X04 Pin IQ - Digital Mode: 0=Digital Input NO normally open,  1=Digital Input NC normally closed, 2=Digital Output, 3=Static On, 4=Not supported.Line = 0; Port X04 Pin IQ - Digital Mode: 0=Digital Input NO normally open,  1=Digital Input NC normally closed, 2=Digital Output, 3=Static On, 4=Not supported.CompleteAccess = False; Port X04 Pin IQ - DI Filter Time: 0=no Filter, 30=3ms, 150=15ms, 200=20ms.Index = 16#2130; Port X04 Pin IQ - DI Filter Time: 0=no Filter, 30=3ms, 150=15ms, 200=20ms.Subindex = 16#05; Port X04 Pin IQ - DI Filter Time: 0=no Filter, 30=3ms, 150=15ms, 200=20ms.Value = 0; Port X04 Pin IQ - DI Filter Time: 0=no Filter, 30=3ms, 150=15ms, 200=20ms.Size = 8; Port X04 Pin IQ - DI Filter Time: 0=no Filter, 30=3ms, 150=15ms, 200=20ms.AbortIfError = FALSE; Port X04 Pin IQ - DI Filter Time: 0=no Filter, 30=3ms, 150=15ms, 200=20ms.JumpToLine = FALSE; Port X04 Pin IQ - DI Filter Time: 0=no Filter, 30=3ms, 150=15ms, 200=20ms.Line = 0; Port X04 Pin IQ - DI Filter Time: 0=no Filter, 30=3ms, 150=15ms, 200=20ms.CompleteAccess = False; Port X05 Pin CQ - DI Invert: false=Digital Input NO normally open,  true=Digital Input NC normally closed.Index = 16#2140; Port X05 Pin CQ - DI Invert: false=Digital Input NO normally open,  true=Digital Input NC normally closed.Subindex = 16#01; Port X05 Pin CQ - DI Invert: false=Digital Input NO normally open,  true=Digital Input NC normally closed.Value = 0; Port X05 Pin CQ - DI Invert: false=Digital Input NO normally open,  true=Digital Input NC normally closed.Size = 8; Port X05 Pin CQ - DI Invert: false=Digital Input NO normally open,  true=Digital Input NC normally closed.AbortIfError = FALSE; Port X05 Pin CQ - DI Invert: false=Digital Input NO normally open,  true=Digital Input NC normally closed.JumpToLine = FALSE; Port X05 Pin CQ - DI Invert: false=Digital Input NO normally open,  true=Digital Input NC normally closed.Line = 0; Port X05 Pin CQ - DI Invert: false=Digital Input NO normally open,  true=Digital Input NC normally closed.CompleteAccess = False; Port X05 Pin CQ - DI Filter Time: 0=no Filter, 30=3ms, 150=15ms, 200=20ms.Index = 16#2140;
            Port X05 Pin CQ - DI Filter Time: 0=no Filter, 30=3ms, 150=15ms, 200=20ms.Subindex = 16#02; Port X05 Pin CQ - DI Filter Time: 0=no Filter, 30=3ms, 150=15ms, 200=20ms.Value = 0; Port X05 Pin CQ - DI Filter Time: 0=no Filter, 30=3ms, 150=15ms, 200=20ms.Size = 8; Port X05 Pin CQ - DI Filter Time: 0=no Filter, 30=3ms, 150=15ms, 200=20ms.AbortIfError = FALSE; Port X05 Pin CQ - DI Filter Time: 0=no Filter, 30=3ms, 150=15ms, 200=20ms.JumpToLine = FALSE; Port X05 Pin CQ - DI Filter Time: 0=no Filter, 30=3ms, 150=15ms, 200=20ms.Line = 0; Port X05 Pin CQ - DI Filter Time: 0=no Filter, 30=3ms, 150=15ms, 200=20ms.CompleteAccess = False; Port X05 Pin CQ - DO Static On: false=off, true=on.Index = 16#2140; Port X05 Pin CQ - DO Static On: false=off, true=on.Subindex = 16#03; Port X05 Pin CQ - DO Static On: false=off, true=on.Value = 0; Port X05 Pin CQ - DO Static On: false=off, true=on.Size = 8; Port X05 Pin CQ - DO Static On: false=off, true=on.AbortIfError = FALSE; Port X05 Pin CQ - DO Static On: false=off, true=on.JumpToLine = FALSE; Port X05 Pin CQ - DO Static On: false=off, true=on.Line = 0; Port X05 Pin CQ - DO Static On: false=off, true=on.CompleteAccess = False; Port X05 Pin IQ - Digital Mode: 0=Digital Input NO normally open,  1=Digital Input NC normally closed, 2=Digital Output, 3=Static On, 4=Not supported.Index = 16#2140; Port X05 Pin IQ - Digital Mode: 0=Digital Input NO normally open,  1=Digital Input NC normally closed, 2=Digital Output, 3=Static On, 4=Not supported.Subindex = 16#04; Port X05 Pin IQ - Digital Mode: 0=Digital Input NO normally open,  1=Digital Input NC normally closed, 2=Digital Output, 3=Static On, 4=Not supported.Value = 4; Port X05 Pin IQ - Digital Mode: 0=Digital Input NO normally open,  1=Digital Input NC normally closed, 2=Digital Output, 3=Static On, 4=Not supported.Size = 8; Port X05 Pin IQ - Digital Mode: 0=Digital Input NO normally open,  1=Digital Input NC normally closed, 2=Digital Output, 3=Static On, 4=Not supported.AbortIfError = FALSE; Port X05 Pin IQ - Digital Mode: 0=Digital Input NO normally open,  1=Digital Input NC normally closed, 2=Digital Output, 3=Static On, 4=Not supported.JumpToLine = FALSE; Port X05 Pin IQ - Digital Mode: 0=Digital Input NO normally open,  1=Digital Input NC normally closed, 2=Digital Output, 3=Static On, 4=Not supported.Line = 0; Port X05 Pin IQ - Digital Mode: 0=Digital Input NO normally open,  1=Digital Input NC normally closed, 2=Digital Output, 3=Static On, 4=Not supported.CompleteAccess = False; Port X05 Pin IQ - DI Filter Time: 0=no Filter, 30=3ms, 150=15ms, 200=20ms.Index = 16#2140; Port X05 Pin IQ - DI Filter Time: 0=no Filter, 30=3ms, 150=15ms, 200=20ms.Subindex = 16#05; Port X05 Pin IQ - DI Filter Time: 0=no Filter, 30=3ms, 150=15ms, 200=20ms.Value = 0; Port X05 Pin IQ - DI Filter Time: 0=no Filter, 30=3ms, 150=15ms, 200=20ms.Size = 8; Port X05 Pin IQ - DI Filter Time: 0=no Filter, 30=3ms, 150=15ms, 200=20ms.AbortIfError = FALSE; Port X05 Pin IQ - DI Filter Time: 0=no Filter, 30=3ms, 150=15ms, 200=20ms.JumpToLine = FALSE; Port X05 Pin IQ - DI Filter Time: 0=no Filter, 30=3ms, 150=15ms, 200=20ms.Line = 0; Port X05 Pin IQ - DI Filter Time: 0=no Filter, 30=3ms, 150=15ms, 200=20ms.CompleteAccess = False; Port X06 Pin CQ - DI Invert: false=Digital Input NO normally open,  true=Digital Input NC normally closed.Index = 16#2150; Port X06 Pin CQ - DI Invert: false=Digital Input NO normally open,  true=Digital Input NC normally closed.Subindex = 16#01; Port X06 Pin CQ - DI Invert: false=Digital Input NO normally open,  true=Digital Input NC normally closed.Value = 0; Port X06 Pin CQ - DI Invert: false=Digital Input NO normally open,  true=Digital Input NC normally closed.Size = 8; Port X06 Pin CQ - DI Invert: false=Digital Input NO normally open,  true=Digital Input NC normally closed.AbortIfError = FALSE; Port X06 Pin CQ - DI Invert: false=Digital Input NO normally open,  true=Digital Input NC normally closed.JumpToLine = FALSE; Port X06 Pin CQ - DI Invert: false=Digital Input NO normally open,  true=Digital Input NC normally closed.Line = 0; Port X06 Pin CQ - DI Invert: false=Digital Input NO normally open,  true=Digital Input NC normally closed.CompleteAccess = False; Port X06 Pin CQ - DI Filter Time: 0=no Filter, 30=3ms, 150=15ms, 200=20ms.Index = 16#2150;
            Port X06 Pin CQ - DI Filter Time: 0=no Filter, 30=3ms, 150=15ms, 200=20ms.Subindex = 16#02; Port X06 Pin CQ - DI Filter Time: 0=no Filter, 30=3ms, 150=15ms, 200=20ms.Value = 0; Port X06 Pin CQ - DI Filter Time: 0=no Filter, 30=3ms, 150=15ms, 200=20ms.Size = 8; Port X06 Pin CQ - DI Filter Time: 0=no Filter, 30=3ms, 150=15ms, 200=20ms.AbortIfError = FALSE; Port X06 Pin CQ - DI Filter Time: 0=no Filter, 30=3ms, 150=15ms, 200=20ms.JumpToLine = FALSE; Port X06 Pin CQ - DI Filter Time: 0=no Filter, 30=3ms, 150=15ms, 200=20ms.Line = 0; Port X06 Pin CQ - DI Filter Time: 0=no Filter, 30=3ms, 150=15ms, 200=20ms.CompleteAccess = False; Port X06 Pin CQ - DO Static On: false=off, true=on.Index = 16#2150; Port X06 Pin CQ - DO Static On: false=off, true=on.Subindex = 16#03; Port X06 Pin CQ - DO Static On: false=off, true=on.Value = 0; Port X06 Pin CQ - DO Static On: false=off, true=on.Size = 8; Port X06 Pin CQ - DO Static On: false=off, true=on.AbortIfError = FALSE; Port X06 Pin CQ - DO Static On: false=off, true=on.JumpToLine = FALSE; Port X06 Pin CQ - DO Static On: false=off, true=on.Line = 0; Port X06 Pin CQ - DO Static On: false=off, true=on.CompleteAccess = False; Port X06 Pin IQ - Digital Mode: 0=Digital Input NO normally open,  1=Digital Input NC normally closed, 2=Digital Output, 3=Static On, 4=Not supported.Index = 16#2150; Port X06 Pin IQ - Digital Mode: 0=Digital Input NO normally open,  1=Digital Input NC normally closed, 2=Digital Output, 3=Static On, 4=Not supported.Subindex = 16#04; Port X06 Pin IQ - Digital Mode: 0=Digital Input NO normally open,  1=Digital Input NC normally closed, 2=Digital Output, 3=Static On, 4=Not supported.Value = 4; Port X06 Pin IQ - Digital Mode: 0=Digital Input NO normally open,  1=Digital Input NC normally closed, 2=Digital Output, 3=Static On, 4=Not supported.Size = 8; Port X06 Pin IQ - Digital Mode: 0=Digital Input NO normally open,  1=Digital Input NC normally closed, 2=Digital Output, 3=Static On, 4=Not supported.AbortIfError = FALSE; Port X06 Pin IQ - Digital Mode: 0=Digital Input NO normally open,  1=Digital Input NC normally closed, 2=Digital Output, 3=Static On, 4=Not supported.JumpToLine = FALSE; Port X06 Pin IQ - Digital Mode: 0=Digital Input NO normally open,  1=Digital Input NC normally closed, 2=Digital Output, 3=Static On, 4=Not supported.Line = 0; Port X06 Pin IQ - Digital Mode: 0=Digital Input NO normally open,  1=Digital Input NC normally closed, 2=Digital Output, 3=Static On, 4=Not supported.CompleteAccess = False; Port X06 Pin IQ - DI Filter Time: 0=no Filter, 30=3ms, 150=15ms, 200=20ms.Index = 16#2150; Port X06 Pin IQ - DI Filter Time: 0=no Filter, 30=3ms, 150=15ms, 200=20ms.Subindex = 16#05; Port X06 Pin IQ - DI Filter Time: 0=no Filter, 30=3ms, 150=15ms, 200=20ms.Value = 0; Port X06 Pin IQ - DI Filter Time: 0=no Filter, 30=3ms, 150=15ms, 200=20ms.Size = 8; Port X06 Pin IQ - DI Filter Time: 0=no Filter, 30=3ms, 150=15ms, 200=20ms.AbortIfError = FALSE; Port X06 Pin IQ - DI Filter Time: 0=no Filter, 30=3ms, 150=15ms, 200=20ms.JumpToLine = FALSE; Port X06 Pin IQ - DI Filter Time: 0=no Filter, 30=3ms, 150=15ms, 200=20ms.Line = 0; Port X06 Pin IQ - DI Filter Time: 0=no Filter, 30=3ms, 150=15ms, 200=20ms.CompleteAccess = False; Port X07 Pin CQ - DI Invert: false=Digital Input NO normally open,  true=Digital Input NC normally closed.Index = 16#2160; Port X07 Pin CQ - DI Invert: false=Digital Input NO normally open,  true=Digital Input NC normally closed.Subindex = 16#01; Port X07 Pin CQ - DI Invert: false=Digital Input NO normally open,  true=Digital Input NC normally closed.Value = 0; Port X07 Pin CQ - DI Invert: false=Digital Input NO normally open,  true=Digital Input NC normally closed.Size = 8; Port X07 Pin CQ - DI Invert: false=Digital Input NO normally open,  true=Digital Input NC normally closed.AbortIfError = FALSE; Port X07 Pin CQ - DI Invert: false=Digital Input NO normally open,  true=Digital Input NC normally closed.JumpToLine = FALSE; Port X07 Pin CQ - DI Invert: false=Digital Input NO normally open,  true=Digital Input NC normally closed.Line = 0; Port X07 Pin CQ - DI Invert: false=Digital Input NO normally open,  true=Digital Input NC normally closed.CompleteAccess = False; Port X07 Pin CQ - DI Filter Time: 0=no Filter, 30=3ms, 150=15ms, 200=20ms.Index = 16#2160;
            Port X07 Pin CQ - DI Filter Time: 0=no Filter, 30=3ms, 150=15ms, 200=20ms.Subindex = 16#02; Port X07 Pin CQ - DI Filter Time: 0=no Filter, 30=3ms, 150=15ms, 200=20ms.Value = 0; Port X07 Pin CQ - DI Filter Time: 0=no Filter, 30=3ms, 150=15ms, 200=20ms.Size = 8; Port X07 Pin CQ - DI Filter Time: 0=no Filter, 30=3ms, 150=15ms, 200=20ms.AbortIfError = FALSE; Port X07 Pin CQ - DI Filter Time: 0=no Filter, 30=3ms, 150=15ms, 200=20ms.JumpToLine = FALSE; Port X07 Pin CQ - DI Filter Time: 0=no Filter, 30=3ms, 150=15ms, 200=20ms.Line = 0; Port X07 Pin CQ - DI Filter Time: 0=no Filter, 30=3ms, 150=15ms, 200=20ms.CompleteAccess = False; Port X07 Pin CQ - DO Static On: false=off, true=on.Index = 16#2160; Port X07 Pin CQ - DO Static On: false=off, true=on.Subindex = 16#03; Port X07 Pin CQ - DO Static On: false=off, true=on.Value = 0; Port X07 Pin CQ - DO Static On: false=off, true=on.Size = 8; Port X07 Pin CQ - DO Static On: false=off, true=on.AbortIfError = FALSE; Port X07 Pin CQ - DO Static On: false=off, true=on.JumpToLine = FALSE; Port X07 Pin CQ - DO Static On: false=off, true=on.Line = 0; Port X07 Pin CQ - DO Static On: false=off, true=on.CompleteAccess = False; Port X07 Pin IQ - Digital Mode: 0=Digital Input NO normally open,  1=Digital Input NC normally closed, 2=Digital Output, 3=Static On, 4=Not supported.Index = 16#2160; Port X07 Pin IQ - Digital Mode: 0=Digital Input NO normally open,  1=Digital Input NC normally closed, 2=Digital Output, 3=Static On, 4=Not supported.Subindex = 16#04; Port X07 Pin IQ - Digital Mode: 0=Digital Input NO normally open,  1=Digital Input NC normally closed, 2=Digital Output, 3=Static On, 4=Not supported.Value = 4; Port X07 Pin IQ - Digital Mode: 0=Digital Input NO normally open,  1=Digital Input NC normally closed, 2=Digital Output, 3=Static On, 4=Not supported.Size = 8; Port X07 Pin IQ - Digital Mode: 0=Digital Input NO normally open,  1=Digital Input NC normally closed, 2=Digital Output, 3=Static On, 4=Not supported.AbortIfError = FALSE; Port X07 Pin IQ - Digital Mode: 0=Digital Input NO normally open,  1=Digital Input NC normally closed, 2=Digital Output, 3=Static On, 4=Not supported.JumpToLine = FALSE; Port X07 Pin IQ - Digital Mode: 0=Digital Input NO normally open,  1=Digital Input NC normally closed, 2=Digital Output, 3=Static On, 4=Not supported.Line = 0; Port X07 Pin IQ - Digital Mode: 0=Digital Input NO normally open,  1=Digital Input NC normally closed, 2=Digital Output, 3=Static On, 4=Not supported.CompleteAccess = False; Port X07 Pin IQ - DI Filter Time: 0=no Filter, 30=3ms, 150=15ms, 200=20ms.Index = 16#2160; Port X07 Pin IQ - DI Filter Time: 0=no Filter, 30=3ms, 150=15ms, 200=20ms.Subindex = 16#05; Port X07 Pin IQ - DI Filter Time: 0=no Filter, 30=3ms, 150=15ms, 200=20ms.Value = 0; Port X07 Pin IQ - DI Filter Time: 0=no Filter, 30=3ms, 150=15ms, 200=20ms.Size = 8; Port X07 Pin IQ - DI Filter Time: 0=no Filter, 30=3ms, 150=15ms, 200=20ms.AbortIfError = FALSE; Port X07 Pin IQ - DI Filter Time: 0=no Filter, 30=3ms, 150=15ms, 200=20ms.JumpToLine = FALSE; Port X07 Pin IQ - DI Filter Time: 0=no Filter, 30=3ms, 150=15ms, 200=20ms.Line = 0; Port X07 Pin IQ - DI Filter Time: 0=no Filter, 30=3ms, 150=15ms, 200=20ms.CompleteAccess = False; Port X08 Pin CQ - DI Invert: false=Digital Input NO normally open,  true=Digital Input NC normally closed.Index = 16#2170; Port X08 Pin CQ - DI Invert: false=Digital Input NO normally open,  true=Digital Input NC normally closed.Subindex = 16#01; Port X08 Pin CQ - DI Invert: false=Digital Input NO normally open,  true=Digital Input NC normally closed.Value = 0; Port X08 Pin CQ - DI Invert: false=Digital Input NO normally open,  true=Digital Input NC normally closed.Size = 8; Port X08 Pin CQ - DI Invert: false=Digital Input NO normally open,  true=Digital Input NC normally closed.AbortIfError = FALSE; Port X08 Pin CQ - DI Invert: false=Digital Input NO normally open,  true=Digital Input NC normally closed.JumpToLine = FALSE; Port X08 Pin CQ - DI Invert: false=Digital Input NO normally open,  true=Digital Input NC normally closed.Line = 0; Port X08 Pin CQ - DI Invert: false=Digital Input NO normally open,  true=Digital Input NC normally closed.CompleteAccess = False; Port X08 Pin CQ - DI Filter Time: 0=no Filter, 30=3ms, 150=15ms, 200=20ms.Index = 16#2170;
            Port X08 Pin CQ - DI Filter Time: 0=no Filter, 30=3ms, 150=15ms, 200=20ms.Subindex = 16#02; Port X08 Pin CQ - DI Filter Time: 0=no Filter, 30=3ms, 150=15ms, 200=20ms.Value = 0; Port X08 Pin CQ - DI Filter Time: 0=no Filter, 30=3ms, 150=15ms, 200=20ms.Size = 8; Port X08 Pin CQ - DI Filter Time: 0=no Filter, 30=3ms, 150=15ms, 200=20ms.AbortIfError = FALSE; Port X08 Pin CQ - DI Filter Time: 0=no Filter, 30=3ms, 150=15ms, 200=20ms.JumpToLine = FALSE; Port X08 Pin CQ - DI Filter Time: 0=no Filter, 30=3ms, 150=15ms, 200=20ms.Line = 0; Port X08 Pin CQ - DI Filter Time: 0=no Filter, 30=3ms, 150=15ms, 200=20ms.CompleteAccess = False; Port X08 Pin CQ - DO Static On: false=off, true=on.Index = 16#2170; Port X08 Pin CQ - DO Static On: false=off, true=on.Subindex = 16#03; Port X08 Pin CQ - DO Static On: false=off, true=on.Value = 0; Port X08 Pin CQ - DO Static On: false=off, true=on.Size = 8; Port X08 Pin CQ - DO Static On: false=off, true=on.AbortIfError = FALSE; Port X08 Pin CQ - DO Static On: false=off, true=on.JumpToLine = FALSE; Port X08 Pin CQ - DO Static On: false=off, true=on.Line = 0; Port X08 Pin CQ - DO Static On: false=off, true=on.CompleteAccess = False; Port X08 Pin IQ - Digital Mode: 0=Digital Input NO normally open,  1=Digital Input NC normally closed, 2=Digital Output, 3=Static On, 4=Not supported.Index = 16#2170; Port X08 Pin IQ - Digital Mode: 0=Digital Input NO normally open,  1=Digital Input NC normally closed, 2=Digital Output, 3=Static On, 4=Not supported.Subindex = 16#04; Port X08 Pin IQ - Digital Mode: 0=Digital Input NO normally open,  1=Digital Input NC normally closed, 2=Digital Output, 3=Static On, 4=Not supported.Value = 4; Port X08 Pin IQ - Digital Mode: 0=Digital Input NO normally open,  1=Digital Input NC normally closed, 2=Digital Output, 3=Static On, 4=Not supported.Size = 8; Port X08 Pin IQ - Digital Mode: 0=Digital Input NO normally open,  1=Digital Input NC normally closed, 2=Digital Output, 3=Static On, 4=Not supported.AbortIfError = FALSE; Port X08 Pin IQ - Digital Mode: 0=Digital Input NO normally open,  1=Digital Input NC normally closed, 2=Digital Output, 3=Static On, 4=Not supported.JumpToLine = FALSE; Port X08 Pin IQ - Digital Mode: 0=Digital Input NO normally open,  1=Digital Input NC normally closed, 2=Digital Output, 3=Static On, 4=Not supported.Line = 0; Port X08 Pin IQ - Digital Mode: 0=Digital Input NO normally open,  1=Digital Input NC normally closed, 2=Digital Output, 3=Static On, 4=Not supported.CompleteAccess = False; Port X08 Pin IQ - DI Filter Time: 0=no Filter, 30=3ms, 150=15ms, 200=20ms.Index = 16#2170; Port X08 Pin IQ - DI Filter Time: 0=no Filter, 30=3ms, 150=15ms, 200=20ms.Subindex = 16#05; Port X08 Pin IQ - DI Filter Time: 0=no Filter, 30=3ms, 150=15ms, 200=20ms.Value = 0; Port X08 Pin IQ - DI Filter Time: 0=no Filter, 30=3ms, 150=15ms, 200=20ms.Size = 8; Port X08 Pin IQ - DI Filter Time: 0=no Filter, 30=3ms, 150=15ms, 200=20ms.AbortIfError = FALSE; Port X08 Pin IQ - DI Filter Time: 0=no Filter, 30=3ms, 150=15ms, 200=20ms.JumpToLine = FALSE; Port X08 Pin IQ - DI Filter Time: 0=no Filter, 30=3ms, 150=15ms, 200=20ms.Line = 0; Port X08 Pin IQ - DI Filter Time: 0=no Filter, 30=3ms, 150=15ms, 200=20ms.CompleteAccess = False; RxTxPdo.NumberofExcludes = 0; RxTxPdo.NumberofEntries = 1; RxTxPdo.Index = 16#1610; RxTxPdo.Fixed = True; RxTxPdo.Mandatory = True; RxTxPdo.Virtual = False; RxTxPdo.Sm = 2; RxTxPdo.Su = 2; RxTxPdo.Name = 'RxPDO Mapping of Digital Outputs';
            RxTxPdo.DependOnSlot = False; RxTxPdo.DependOnSlotGroup = False; RxTxPdo.OverwrittenByModule = False; PD (I/Q Pin2).Index = 16#3001; PD (I/Q Pin2).SubIndex = 1; PD (I/Q Pin2).Size = 16; PD (I/Q Pin2).Offset = 0; PD (I/Q Pin2).DependOnSlot = False; PD (I/Q Pin2).DependOnSlotGroup = False; RxTxPdo.NumberofExcludes = 0; RxTxPdo.NumberofEntries = 8; RxTxPdo.Index = 16#1600; RxTxPdo.Fixed = False; RxTxPdo.Mandatory = False; RxTxPdo.Virtual = False; RxTxPdo.Sm = 2; RxTxPdo.Su = 0; RxTxPdo.Name = 'RxPDO'; RxTxPdo.DependOnSlot = True; RxTxPdo.DependOnSlotGroup = False; RxTxPdo.OverwrittenByModule = True; output byte 0.Index = 16#7000; output byte 0.SubIndex = 1; output byte 0.Size = 8; output byte 0.Offset = 0; output byte 0.DependOnSlot = True; output byte 0.DependOnSlotGroup = False; output byte 1.Index = 16#7000; output byte 1.SubIndex = 2; output byte 1.Size = 8; output byte 1.Offset = 0; output byte 1.DependOnSlot = True; output byte 1.DependOnSlotGroup = False; output byte 2.Index = 16#7000; output byte 2.SubIndex = 3; output byte 2.Size = 8; output byte 2.Offset = 0; output byte 2.DependOnSlot = True; output byte 2.DependOnSlotGroup = False; output byte 3.Index = 16#7000;
            output byte 3.SubIndex = 4; output byte 3.Size = 8; output byte 3.Offset = 0; output byte 3.DependOnSlot = True; output byte 3.DependOnSlotGroup = False; output byte 4.Index = 16#7000; output byte 4.SubIndex = 5; output byte 4.Size = 8; output byte 4.Offset = 0; output byte 4.DependOnSlot = True; output byte 4.DependOnSlotGroup = False; output byte 5.Index = 16#7000; output byte 5.SubIndex = 6; output byte 5.Size = 8; output byte 5.Offset = 0; output byte 5.DependOnSlot = True; output byte 5.DependOnSlotGroup = False; output byte 6.Index = 16#7000; output byte 6.SubIndex = 7; output byte 6.Size = 8; output byte 6.Offset = 0; output byte 6.DependOnSlot = True; output byte 6.DependOnSlotGroup = False; output byte 7.Index = 16#7000; output byte 7.SubIndex = 8; output byte 7.Size = 8; output byte 7.Offset = 0; output byte 7.DependOnSlot = True; output byte 7.DependOnSlotGroup = False; RxTxPdo.NumberofExcludes = 0; RxTxPdo.NumberofEntries = 1; RxTxPdo.Index = 16#1601; RxTxPdo.Fixed = False; RxTxPdo.Mandatory = False; RxTxPdo.Virtual = False; RxTxPdo.Sm = 2; RxTxPdo.Su = 0; RxTxPdo.Name = 'RxPDO'; RxTxPdo.DependOnSlot = True; RxTxPdo.DependOnSlotGroup = False;
            RxTxPdo.OverwrittenByModule = True; PD (C/Q Pin4).Index = 16#7010; PD (C/Q Pin4).SubIndex = 1; PD (C/Q Pin4).Size = 8; PD (C/Q Pin4).Offset = 0; PD (C/Q Pin4).DependOnSlot = True; PD (C/Q Pin4).DependOnSlotGroup = False; RxTxPdo.NumberofExcludes = 0; RxTxPdo.NumberofEntries = 2; RxTxPdo.Index = 16#1602; RxTxPdo.Fixed = False; RxTxPdo.Mandatory = False; RxTxPdo.Virtual = False; RxTxPdo.Sm = 2; RxTxPdo.Su = 0; RxTxPdo.Name = 'RxPDO'; RxTxPdo.DependOnSlot = True; RxTxPdo.DependOnSlotGroup = False; RxTxPdo.OverwrittenByModule = True; output byte 0.Index = 16#7020; output byte 0.SubIndex = 1; output byte 0.Size = 8; output byte 0.Offset = 0; output byte 0.DependOnSlot = True; output byte 0.DependOnSlotGroup = False; output byte 1.Index = 16#7020; output byte 1.SubIndex = 2; output byte 1.Size = 8; output byte 1.Offset = 0; output byte 1.DependOnSlot = True; output byte 1.DependOnSlotGroup = False; RxTxPdo.NumberofExcludes = 0; RxTxPdo.NumberofEntries = 1; RxTxPdo.Index = 16#1603; RxTxPdo.Fixed = False; RxTxPdo.Mandatory = False; RxTxPdo.Virtual = False; RxTxPdo.Sm = 2; RxTxPdo.Su = 0; RxTxPdo.Name = 'RxPDO';
            RxTxPdo.DependOnSlot = True; RxTxPdo.DependOnSlotGroup = False; RxTxPdo.OverwrittenByModule = True; PD (C/Q Pin4).Index = 16#7030; PD (C/Q Pin4).SubIndex = 1; PD (C/Q Pin4).Size = 8; PD (C/Q Pin4).Offset = 0; PD (C/Q Pin4).DependOnSlot = True; PD (C/Q Pin4).DependOnSlotGroup = False; RxTxPdo.NumberofExcludes = 0; RxTxPdo.NumberofEntries = 2; RxTxPdo.Index = 16#1604; RxTxPdo.Fixed = False; RxTxPdo.Mandatory = False; RxTxPdo.Virtual = False; RxTxPdo.Sm = 2; RxTxPdo.Su = 0; RxTxPdo.Name = 'RxPDO'; RxTxPdo.DependOnSlot = True; RxTxPdo.DependOnSlotGroup = False; RxTxPdo.OverwrittenByModule = True; output byte 0.Index = 16#7040; output byte 0.SubIndex = 1; output byte 0.Size = 8; output byte 0.Offset = 0; output byte 0.DependOnSlot = True; output byte 0.DependOnSlotGroup = False; output byte 1.Index = 16#7040; output byte 1.SubIndex = 2; output byte 1.Size = 8; output byte 1.Offset = 0; output byte 1.DependOnSlot = True; output byte 1.DependOnSlotGroup = False; RxTxPdo.NumberofExcludes = 0; RxTxPdo.NumberofEntries = 32; RxTxPdo.Index = 16#1606; RxTxPdo.Fixed = False; RxTxPdo.Mandatory = False; RxTxPdo.Virtual = False; RxTxPdo.Sm = 2;
            RxTxPdo.Su = 0; RxTxPdo.Name = 'RxPDO'; RxTxPdo.DependOnSlot = True; RxTxPdo.DependOnSlotGroup = False; RxTxPdo.OverwrittenByModule = True; output byte 0.Index = 16#7060; output byte 0.SubIndex = 1; output byte 0.Size = 8; output byte 0.Offset = 0; output byte 0.DependOnSlot = True; output byte 0.DependOnSlotGroup = False; output byte 1.Index = 16#7060; output byte 1.SubIndex = 2; output byte 1.Size = 8; output byte 1.Offset = 0; output byte 1.DependOnSlot = True; output byte 1.DependOnSlotGroup = False; output byte 2.Index = 16#7060; output byte 2.SubIndex = 3; output byte 2.Size = 8; output byte 2.Offset = 0; output byte 2.DependOnSlot = True; output byte 2.DependOnSlotGroup = False; output byte 3.Index = 16#7060; output byte 3.SubIndex = 4; output byte 3.Size = 8; output byte 3.Offset = 0; output byte 3.DependOnSlot = True; output byte 3.DependOnSlotGroup = False; output byte 4.Index = 16#7060; output byte 4.SubIndex = 5; output byte 4.Size = 8; output byte 4.Offset = 0; output byte 4.DependOnSlot = True; output byte 4.DependOnSlotGroup = False; output byte 5.Index = 16#7060; output byte 5.SubIndex = 6; output byte 5.Size = 8; output byte 5.Offset = 0; output byte 5.DependOnSlot = True;
            output byte 5.DependOnSlotGroup = False; output byte 6.Index = 16#7060; output byte 6.SubIndex = 7; output byte 6.Size = 8; output byte 6.Offset = 0; output byte 6.DependOnSlot = True; output byte 6.DependOnSlotGroup = False; output byte 7.Index = 16#7060; output byte 7.SubIndex = 8; output byte 7.Size = 8; output byte 7.Offset = 0; output byte 7.DependOnSlot = True; output byte 7.DependOnSlotGroup = False; output byte 8.Index = 16#7060; output byte 8.SubIndex = 9; output byte 8.Size = 8; output byte 8.Offset = 0; output byte 8.DependOnSlot = True; output byte 8.DependOnSlotGroup = False; output byte 9.Index = 16#7060; output byte 9.SubIndex = 10; output byte 9.Size = 8; output byte 9.Offset = 0; output byte 9.DependOnSlot = True; output byte 9.DependOnSlotGroup = False; output byte 10.Index = 16#7060; output byte 10.SubIndex = 11; output byte 10.Size = 8; output byte 10.Offset = 0; output byte 10.DependOnSlot = True; output byte 10.DependOnSlotGroup = False; output byte 11.Index = 16#7060; output byte 11.SubIndex = 12; output byte 11.Size = 8; output byte 11.Offset = 0; output byte 11.DependOnSlot = True; output byte 11.DependOnSlotGroup = False; output byte 12.Index = 16#7060; output byte 12.SubIndex = 13; output byte 12.Size = 8;
            output byte 12.Offset = 0; output byte 12.DependOnSlot = True; output byte 12.DependOnSlotGroup = False; output byte 13.Index = 16#7060; output byte 13.SubIndex = 14; output byte 13.Size = 8; output byte 13.Offset = 0; output byte 13.DependOnSlot = True; output byte 13.DependOnSlotGroup = False; output byte 14.Index = 16#7060; output byte 14.SubIndex = 15; output byte 14.Size = 8; output byte 14.Offset = 0; output byte 14.DependOnSlot = True; output byte 14.DependOnSlotGroup = False; output byte 15.Index = 16#7060; output byte 15.SubIndex = 16; output byte 15.Size = 8; output byte 15.Offset = 0; output byte 15.DependOnSlot = True; output byte 15.DependOnSlotGroup = False; output byte 16.Index = 16#7060; output byte 16.SubIndex = 17; output byte 16.Size = 8; output byte 16.Offset = 0; output byte 16.DependOnSlot = True; output byte 16.DependOnSlotGroup = False; output byte 17.Index = 16#7060; output byte 17.SubIndex = 18; output byte 17.Size = 8; output byte 17.Offset = 0; output byte 17.DependOnSlot = True; output byte 17.DependOnSlotGroup = False; output byte 18.Index = 16#7060; output byte 18.SubIndex = 19; output byte 18.Size = 8; output byte 18.Offset = 0; output byte 18.DependOnSlot = True; output byte 18.DependOnSlotGroup = False; output byte 19.Index = 16#7060;
            output byte 19.SubIndex = 20; output byte 19.Size = 8; output byte 19.Offset = 0; output byte 19.DependOnSlot = True; output byte 19.DependOnSlotGroup = False; output byte 20.Index = 16#7060; output byte 20.SubIndex = 21; output byte 20.Size = 8; output byte 20.Offset = 0; output byte 20.DependOnSlot = True; output byte 20.DependOnSlotGroup = False; output byte 21.Index = 16#7060; output byte 21.SubIndex = 22; output byte 21.Size = 8; output byte 21.Offset = 0; output byte 21.DependOnSlot = True; output byte 21.DependOnSlotGroup = False; output byte 22.Index = 16#7060; output byte 22.SubIndex = 23; output byte 22.Size = 8; output byte 22.Offset = 0; output byte 22.DependOnSlot = True; output byte 22.DependOnSlotGroup = False; output byte 23.Index = 16#7060; output byte 23.SubIndex = 24; output byte 23.Size = 8; output byte 23.Offset = 0; output byte 23.DependOnSlot = True; output byte 23.DependOnSlotGroup = False; output byte 24.Index = 16#7060; output byte 24.SubIndex = 25; output byte 24.Size = 8; output byte 24.Offset = 0; output byte 24.DependOnSlot = True; output byte 24.DependOnSlotGroup = False; output byte 25.Index = 16#7060; output byte 25.SubIndex = 26; output byte 25.Size = 8; output byte 25.Offset = 0; output byte 25.DependOnSlot = True;
            output byte 25.DependOnSlotGroup = False; output byte 26.Index = 16#7060; output byte 26.SubIndex = 27; output byte 26.Size = 8; output byte 26.Offset = 0; output byte 26.DependOnSlot = True; output byte 26.DependOnSlotGroup = False; output byte 27.Index = 16#7060; output byte 27.SubIndex = 28; output byte 27.Size = 8; output byte 27.Offset = 0; output byte 27.DependOnSlot = True; output byte 27.DependOnSlotGroup = False; output byte 28.Index = 16#7060; output byte 28.SubIndex = 29; output byte 28.Size = 8; output byte 28.Offset = 0; output byte 28.DependOnSlot = True; output byte 28.DependOnSlotGroup = False; output byte 29.Index = 16#7060; output byte 29.SubIndex = 30; output byte 29.Size = 8; output byte 29.Offset = 0; output byte 29.DependOnSlot = True; output byte 29.DependOnSlotGroup = False; output byte 30.Index = 16#7060; output byte 30.SubIndex = 31; output byte 30.Size = 8; output byte 30.Offset = 0; output byte 30.DependOnSlot = True; output byte 30.DependOnSlotGroup = False; output byte 31.Index = 16#7060; output byte 31.SubIndex = 32; output byte 31.Size = 8; output byte 31.Offset = 0; output byte 31.DependOnSlot = True; output byte 31.DependOnSlotGroup = False; RxTxPdo.NumberofExcludes = 0; RxTxPdo.NumberofEntries = 1; RxTxPdo.Index = 16#1A10;
            RxTxPdo.Fixed = True; RxTxPdo.Mandatory = True; RxTxPdo.Virtual = False; RxTxPdo.Sm = 3; RxTxPdo.Su = 3; RxTxPdo.Name = 'TxPDO Mapping of Digital Inputs'; RxTxPdo.DependOnSlot = False; RxTxPdo.DependOnSlotGroup = False; RxTxPdo.OverwrittenByModule = False; PD (I/Q Pin2 + C/Q Pin4).Index = 16#3000; PD (I/Q Pin2 + C/Q Pin4).SubIndex = 1; PD (I/Q Pin2 + C/Q Pin4).Size = 16; PD (I/Q Pin2 + C/Q Pin4).Offset = 0; PD (I/Q Pin2 + C/Q Pin4).DependOnSlot = False; PD (I/Q Pin2 + C/Q Pin4).DependOnSlotGroup = False; RxTxPdo.NumberofExcludes = 0; RxTxPdo.NumberofEntries = 2; RxTxPdo.Index = 16#1A11; RxTxPdo.Fixed = True; RxTxPdo.Mandatory = True; RxTxPdo.Virtual = False; RxTxPdo.Sm = 3; RxTxPdo.Su = 3; RxTxPdo.Name = 'TxPDO Mapping of New Messages Available'; RxTxPdo.DependOnSlot = False; RxTxPdo.DependOnSlotGroup = False; RxTxPdo.OverwrittenByModule = False; New Message Available Flag.Index = 16#10F3; New Message Available Flag.SubIndex = 4; New Message Available Flag.Size = 1; New Message Available Flag.Offset = 0; New Message Available Flag.DependOnSlot = False; New Message Available Flag.DependOnSlotGroup = False; Dummy.Index = 16#0000; Dummy.SubIndex = 0; Dummy.Size = 7; Dummy.Offset = 0; Dummy.DependOnSlot = False; Dummy.DependOnSlotGroup = False; RxTxPdo.NumberofExcludes = 0;
            RxTxPdo.NumberofEntries = 8; RxTxPdo.Index = 16#1A80; RxTxPdo.Fixed = True; RxTxPdo.Mandatory = True; RxTxPdo.Virtual = False; RxTxPdo.Sm = 3; RxTxPdo.Su = 3; RxTxPdo.Name = 'TxPDO Mapping of Status Data'; RxTxPdo.DependOnSlot = False; RxTxPdo.DependOnSlotGroup = False; RxTxPdo.OverwrittenByModule = False; State of IO-Link Port X01.Index = 16#F100; State of IO-Link Port X01.SubIndex = 1; State of IO-Link Port X01.Size = 8; State of IO-Link Port X01.Offset = 0; State of IO-Link Port X01.DependOnSlot = False; State of IO-Link Port X01.DependOnSlotGroup = False; State of IO-Link Port X02.Index = 16#F100; State of IO-Link Port X02.SubIndex = 2; State of IO-Link Port X02.Size = 8; State of IO-Link Port X02.Offset = 0; State of IO-Link Port X02.DependOnSlot = False; State of IO-Link Port X02.DependOnSlotGroup = False; State of IO-Link Port X03.Index = 16#F100; State of IO-Link Port X03.SubIndex = 3; State of IO-Link Port X03.Size = 8; State of IO-Link Port X03.Offset = 0; State of IO-Link Port X03.DependOnSlot = False; State of IO-Link Port X03.DependOnSlotGroup = False; State of IO-Link Port X04.Index = 16#F100; State of IO-Link Port X04.SubIndex = 4; State of IO-Link Port X04.Size = 8; State of IO-Link Port X04.Offset = 0; State of IO-Link Port X04.DependOnSlot = False; State of IO-Link Port X04.DependOnSlotGroup = False; State of IO-Link Port X05.Index = 16#F100; State of IO-Link Port X05.SubIndex = 5; State of IO-Link Port X05.Size = 8; State of IO-Link Port X05.Offset = 0; State of IO-Link Port X05.DependOnSlot = False;
            State of IO-Link Port X05.DependOnSlotGroup = False; State of IO-Link Port X06.Index = 16#F100; State of IO-Link Port X06.SubIndex = 6; State of IO-Link Port X06.Size = 8; State of IO-Link Port X06.Offset = 0; State of IO-Link Port X06.DependOnSlot = False; State of IO-Link Port X06.DependOnSlotGroup = False; State of IO-Link Port X07.Index = 16#F100; State of IO-Link Port X07.SubIndex = 7; State of IO-Link Port X07.Size = 8; State of IO-Link Port X07.Offset = 0; State of IO-Link Port X07.DependOnSlot = False; State of IO-Link Port X07.DependOnSlotGroup = False; State of IO-Link Port X08.Index = 16#F100; State of IO-Link Port X08.SubIndex = 8; State of IO-Link Port X08.Size = 8; State of IO-Link Port X08.Offset = 0; State of IO-Link Port X08.DependOnSlot = False; State of IO-Link Port X08.DependOnSlotGroup = False; RxTxPdo.NumberofExcludes = 0; RxTxPdo.NumberofEntries = 8; RxTxPdo.Index = 16#1A00; RxTxPdo.Fixed = False; RxTxPdo.Mandatory = False; RxTxPdo.Virtual = False; RxTxPdo.Sm = 3; RxTxPdo.Su = 0; RxTxPdo.Name = 'TxPDO'; RxTxPdo.DependOnSlot = True; RxTxPdo.DependOnSlotGroup = False; RxTxPdo.OverwrittenByModule = True; input byte 0.Index = 16#6000; input byte 0.SubIndex = 1; input byte 0.Size = 8; input byte 0.Offset = 0; input byte 0.DependOnSlot = True; input byte 0.DependOnSlotGroup = False; input byte 1.Index = 16#6000; input byte 1.SubIndex = 2; input byte 1.Size = 8;
            input byte 1.Offset = 0; input byte 1.DependOnSlot = True; input byte 1.DependOnSlotGroup = False; input byte 2.Index = 16#6000; input byte 2.SubIndex = 3; input byte 2.Size = 8; input byte 2.Offset = 0; input byte 2.DependOnSlot = True; input byte 2.DependOnSlotGroup = False; input byte 3.Index = 16#6000; input byte 3.SubIndex = 4; input byte 3.Size = 8; input byte 3.Offset = 0; input byte 3.DependOnSlot = True; input byte 3.DependOnSlotGroup = False; input byte 4.Index = 16#6000; input byte 4.SubIndex = 5; input byte 4.Size = 8; input byte 4.Offset = 0; input byte 4.DependOnSlot = True; input byte 4.DependOnSlotGroup = False; input byte 5.Index = 16#6000; input byte 5.SubIndex = 6; input byte 5.Size = 8; input byte 5.Offset = 0; input byte 5.DependOnSlot = True; input byte 5.DependOnSlotGroup = False; input byte 6.Index = 16#6000; input byte 6.SubIndex = 7; input byte 6.Size = 8; input byte 6.Offset = 0; input byte 6.DependOnSlot = True; input byte 6.DependOnSlotGroup = False; input byte 7.Index = 16#6000; input byte 7.SubIndex = 8; input byte 7.Size = 8; input byte 7.Offset = 0; input byte 7.DependOnSlot = True; input byte 7.DependOnSlotGroup = False; RxTxPdo.NumberofExcludes = 0;
            RxTxPdo.NumberofEntries = 2; RxTxPdo.Index = 16#1A02; RxTxPdo.Fixed = False; RxTxPdo.Mandatory = False; RxTxPdo.Virtual = False; RxTxPdo.Sm = 3; RxTxPdo.Su = 0; RxTxPdo.Name = 'TxPDO'; RxTxPdo.DependOnSlot = True; RxTxPdo.DependOnSlotGroup = False; RxTxPdo.OverwrittenByModule = True; input byte 0.Index = 16#6020; input byte 0.SubIndex = 1; input byte 0.Size = 8; input byte 0.Offset = 0; input byte 0.DependOnSlot = True; input byte 0.DependOnSlotGroup = False; input byte 1.Index = 16#6020; input byte 1.SubIndex = 2; input byte 1.Size = 8; input byte 1.Offset = 0; input byte 1.DependOnSlot = True; input byte 1.DependOnSlotGroup = False; RxTxPdo.NumberofExcludes = 0; RxTxPdo.NumberofEntries = 2; RxTxPdo.Index = 16#1A04; RxTxPdo.Fixed = False; RxTxPdo.Mandatory = False; RxTxPdo.Virtual = False; RxTxPdo.Sm = 3; RxTxPdo.Su = 0; RxTxPdo.Name = 'TxPDO'; RxTxPdo.DependOnSlot = True; RxTxPdo.DependOnSlotGroup = False; RxTxPdo.OverwrittenByModule = True; input byte 0.Index = 16#6040; input byte 0.SubIndex = 1; input byte 0.Size = 8; input byte 0.Offset = 0; input byte 0.DependOnSlot = True;
            input byte 0.DependOnSlotGroup = False; input byte 1.Index = 16#6040; input byte 1.SubIndex = 2; input byte 1.Size = 8; input byte 1.Offset = 0; input byte 1.DependOnSlot = True; input byte 1.DependOnSlotGroup = False; RxTxPdo.NumberofExcludes = 0; RxTxPdo.NumberofEntries = 1; RxTxPdo.Index = 16#1A05; RxTxPdo.Fixed = False; RxTxPdo.Mandatory = False; RxTxPdo.Virtual = False; RxTxPdo.Sm = 3; RxTxPdo.Su = 0; RxTxPdo.Name = 'TxPDO'; RxTxPdo.DependOnSlot = True; RxTxPdo.DependOnSlotGroup = False; RxTxPdo.OverwrittenByModule = True; PD (C/Q Pin4).Index = 16#6050; PD (C/Q Pin4).SubIndex = 1; PD (C/Q Pin4).Size = 8; PD (C/Q Pin4).Offset = 0; PD (C/Q Pin4).DependOnSlot = True; PD (C/Q Pin4).DependOnSlotGroup = False; RxTxPdo.NumberofExcludes = 0; RxTxPdo.NumberofEntries = 32; RxTxPdo.Index = 16#1A06; RxTxPdo.Fixed = False; RxTxPdo.Mandatory = False; RxTxPdo.Virtual = False; RxTxPdo.Sm = 3; RxTxPdo.Su = 0; RxTxPdo.Name = 'TxPDO'; RxTxPdo.DependOnSlot = True; RxTxPdo.DependOnSlotGroup = False; RxTxPdo.OverwrittenByModule = True; input byte 0.Index = 16#6060; input byte 0.SubIndex = 1; input byte 0.Size = 8;
            input byte 0.Offset = 0; input byte 0.DependOnSlot = True; input byte 0.DependOnSlotGroup = False; input byte 1.Index = 16#6060; input byte 1.SubIndex = 2; input byte 1.Size = 8; input byte 1.Offset = 0; input byte 1.DependOnSlot = True; input byte 1.DependOnSlotGroup = False; input byte 2.Index = 16#6060; input byte 2.SubIndex = 3; input byte 2.Size = 8; input byte 2.Offset = 0; input byte 2.DependOnSlot = True; input byte 2.DependOnSlotGroup = False; input byte 3.Index = 16#6060; input byte 3.SubIndex = 4; input byte 3.Size = 8; input byte 3.Offset = 0; input byte 3.DependOnSlot = True; input byte 3.DependOnSlotGroup = False; input byte 4.Index = 16#6060; input byte 4.SubIndex = 5; input byte 4.Size = 8; input byte 4.Offset = 0; input byte 4.DependOnSlot = True; input byte 4.DependOnSlotGroup = False; input byte 5.Index = 16#6060; input byte 5.SubIndex = 6; input byte 5.Size = 8; input byte 5.Offset = 0; input byte 5.DependOnSlot = True; input byte 5.DependOnSlotGroup = False; input byte 6.Index = 16#6060; input byte 6.SubIndex = 7; input byte 6.Size = 8; input byte 6.Offset = 0; input byte 6.DependOnSlot = True; input byte 6.DependOnSlotGroup = False; input byte 7.Index = 16#6060;
            input byte 7.SubIndex = 8; input byte 7.Size = 8; input byte 7.Offset = 0; input byte 7.DependOnSlot = True; input byte 7.DependOnSlotGroup = False; input byte 8.Index = 16#6060; input byte 8.SubIndex = 9; input byte 8.Size = 8; input byte 8.Offset = 0; input byte 8.DependOnSlot = True; input byte 8.DependOnSlotGroup = False; input byte 9.Index = 16#6060; input byte 9.SubIndex = 10; input byte 9.Size = 8; input byte 9.Offset = 0; input byte 9.DependOnSlot = True; input byte 9.DependOnSlotGroup = False; input byte 10.Index = 16#6060; input byte 10.SubIndex = 11; input byte 10.Size = 8; input byte 10.Offset = 0; input byte 10.DependOnSlot = True; input byte 10.DependOnSlotGroup = False; input byte 11.Index = 16#6060; input byte 11.SubIndex = 12; input byte 11.Size = 8; input byte 11.Offset = 0; input byte 11.DependOnSlot = True; input byte 11.DependOnSlotGroup = False; input byte 12.Index = 16#6060; input byte 12.SubIndex = 13; input byte 12.Size = 8; input byte 12.Offset = 0; input byte 12.DependOnSlot = True; input byte 12.DependOnSlotGroup = False; input byte 13.Index = 16#6060; input byte 13.SubIndex = 14; input byte 13.Size = 8; input byte 13.Offset = 0; input byte 13.DependOnSlot = True;
            input byte 13.DependOnSlotGroup = False; input byte 14.Index = 16#6060; input byte 14.SubIndex = 15; input byte 14.Size = 8; input byte 14.Offset = 0; input byte 14.DependOnSlot = True; input byte 14.DependOnSlotGroup = False; input byte 15.Index = 16#6060; input byte 15.SubIndex = 16; input byte 15.Size = 8; input byte 15.Offset = 0; input byte 15.DependOnSlot = True; input byte 15.DependOnSlotGroup = False; input byte 16.Index = 16#6060; input byte 16.SubIndex = 17; input byte 16.Size = 8; input byte 16.Offset = 0; input byte 16.DependOnSlot = True; input byte 16.DependOnSlotGroup = False; input byte 17.Index = 16#6060; input byte 17.SubIndex = 18; input byte 17.Size = 8; input byte 17.Offset = 0; input byte 17.DependOnSlot = True; input byte 17.DependOnSlotGroup = False; input byte 18.Index = 16#6060; input byte 18.SubIndex = 19; input byte 18.Size = 8; input byte 18.Offset = 0; input byte 18.DependOnSlot = True; input byte 18.DependOnSlotGroup = False; input byte 19.Index = 16#6060; input byte 19.SubIndex = 20; input byte 19.Size = 8; input byte 19.Offset = 0; input byte 19.DependOnSlot = True; input byte 19.DependOnSlotGroup = False; input byte 20.Index = 16#6060; input byte 20.SubIndex = 21; input byte 20.Size = 8;
            input byte 20.Offset = 0; input byte 20.DependOnSlot = True; input byte 20.DependOnSlotGroup = False; input byte 21.Index = 16#6060; input byte 21.SubIndex = 22; input byte 21.Size = 8; input byte 21.Offset = 0; input byte 21.DependOnSlot = True; input byte 21.DependOnSlotGroup = False; input byte 22.Index = 16#6060; input byte 22.SubIndex = 23; input byte 22.Size = 8; input byte 22.Offset = 0; input byte 22.DependOnSlot = True; input byte 22.DependOnSlotGroup = False; input byte 23.Index = 16#6060; input byte 23.SubIndex = 24; input byte 23.Size = 8; input byte 23.Offset = 0; input byte 23.DependOnSlot = True; input byte 23.DependOnSlotGroup = False; input byte 24.Index = 16#6060; input byte 24.SubIndex = 25; input byte 24.Size = 8; input byte 24.Offset = 0; input byte 24.DependOnSlot = True; input byte 24.DependOnSlotGroup = False; input byte 25.Index = 16#6060; input byte 25.SubIndex = 26; input byte 25.Size = 8; input byte 25.Offset = 0; input byte 25.DependOnSlot = True; input byte 25.DependOnSlotGroup = False; input byte 26.Index = 16#6060; input byte 26.SubIndex = 27; input byte 26.Size = 8; input byte 26.Offset = 0; input byte 26.DependOnSlot = True; input byte 26.DependOnSlotGroup = False; input byte 27.Index = 16#6060;
            input byte 27.SubIndex = 28; input byte 27.Size = 8; input byte 27.Offset = 0; input byte 27.DependOnSlot = True; input byte 27.DependOnSlotGroup = False; input byte 28.Index = 16#6060; input byte 28.SubIndex = 29; input byte 28.Size = 8; input byte 28.Offset = 0; input byte 28.DependOnSlot = True; input byte 28.DependOnSlotGroup = False; input byte 29.Index = 16#6060; input byte 29.SubIndex = 30; input byte 29.Size = 8; input byte 29.Offset = 0; input byte 29.DependOnSlot = True; input byte 29.DependOnSlotGroup = False; input byte 30.Index = 16#6060; input byte 30.SubIndex = 31; input byte 30.Size = 8; input byte 30.Offset = 0; input byte 30.DependOnSlot = True; input byte 30.DependOnSlotGroup = False; input byte 31.Index = 16#6060; input byte 31.SubIndex = 32; input byte 31.Size = 8; input byte 31.Offset = 0; input byte 31.DependOnSlot = True; input byte 31.DependOnSlotGroup = False; RxTxPdo.NumberofExcludes = 0; RxTxPdo.NumberofEntries = 1; RxTxPdo.Index = 16#1A07; RxTxPdo.Fixed = False; RxTxPdo.Mandatory = False; RxTxPdo.Virtual = False; RxTxPdo.Sm = 3; RxTxPdo.Su = 0; RxTxPdo.Name = 'TxPDO'; RxTxPdo.DependOnSlot = True; RxTxPdo.DependOnSlotGroup = False;
            RxTxPdo.OverwrittenByModule = True; PD (C/Q Pin4).Index = 16#6070; PD (C/Q Pin4).SubIndex = 1; PD (C/Q Pin4).Size = 8; PD (C/Q Pin4).Offset = 0; PD (C/Q Pin4).DependOnSlot = True; PD (C/Q Pin4).DependOnSlotGroup = False; PD (I/Q Pin2).Name = 'PD (I/Q Pin2)'; PD (I/Q Pin2).DataType = 'UINT'; PD (I/Q Pin2).Default = ''; PD (I/Q Pin2).Comment = ''; output byte 0.Name = 'output byte 0'; output byte 0.DataType = 'USINT'; output byte 0.Default = ''; output byte 0.Comment = ''; output byte 1.Name = 'output byte 1'; output byte 1.DataType = 'USINT'; output byte 1.Default = ''; output byte 1.Comment = ''; output byte 2.Name = 'output byte 2'; output byte 2.DataType = 'USINT'; output byte 2.Default = ''; output byte 2.Comment = ''; output byte 3.Name = 'output byte 3'; output byte 3.DataType = 'USINT'; output byte 3.Default = ''; output byte 3.Comment = ''; output byte 4.Name = 'output byte 4'; output byte 4.DataType = 'USINT'; output byte 4.Default = ''; output byte 4.Comment = ''; output byte 5.Name = 'output byte 5'; output byte 5.DataType = 'USINT'; output byte 5.Default = ''; output byte 5.Comment = ''; output byte 6.Name = 'output byte 6'; output byte 6.DataType = 'USINT'; output byte 6.Default = ''; output byte 6.Comment = ''; output byte 7.Name = 'output byte 7';
            output byte 7.DataType = 'USINT'; output byte 7.Default = ''; output byte 7.Comment = ''; PD (C/Q Pin4).Name = 'PD (C/Q Pin4)'; PD (C/Q Pin4).DataType = 'USINT'; PD (C/Q Pin4).Default = ''; PD (C/Q Pin4).Comment = ''; output byte 0.Name = 'output byte 0'; output byte 0.DataType = 'USINT'; output byte 0.Default = ''; output byte 0.Comment = ''; output byte 1.Name = 'output byte 1'; output byte 1.DataType = 'USINT'; output byte 1.Default = ''; output byte 1.Comment = ''; PD (C/Q Pin4).Name = 'PD (C/Q Pin4)'; PD (C/Q Pin4).DataType = 'USINT'; PD (C/Q Pin4).Default = ''; PD (C/Q Pin4).Comment = ''; output byte 0.Name = 'output byte 0'; output byte 0.DataType = 'USINT'; output byte 0.Default = ''; output byte 0.Comment = ''; output byte 1.Name = 'output byte 1'; output byte 1.DataType = 'USINT'; output byte 1.Default = ''; output byte 1.Comment = ''; output byte 0.Name = 'output byte 0'; output byte 0.DataType = 'USINT'; output byte 0.Default = ''; output byte 0.Comment = ''; output byte 1.Name = 'output byte 1'; output byte 1.DataType = 'USINT'; output byte 1.Default = ''; output byte 1.Comment = ''; output byte 2.Name = 'output byte 2'; output byte 2.DataType = 'USINT'; output byte 2.Default = ''; output byte 2.Comment = ''; output byte 3.Name = 'output byte 3';
            output byte 3.DataType = 'USINT'; output byte 3.Default = ''; output byte 3.Comment = ''; output byte 4.Name = 'output byte 4'; output byte 4.DataType = 'USINT'; output byte 4.Default = ''; output byte 4.Comment = ''; output byte 5.Name = 'output byte 5'; output byte 5.DataType = 'USINT'; output byte 5.Default = ''; output byte 5.Comment = ''; output byte 6.Name = 'output byte 6'; output byte 6.DataType = 'USINT'; output byte 6.Default = ''; output byte 6.Comment = ''; output byte 7.Name = 'output byte 7'; output byte 7.DataType = 'USINT'; output byte 7.Default = ''; output byte 7.Comment = ''; output byte 8.Name = 'output byte 8'; output byte 8.DataType = 'USINT'; output byte 8.Default = ''; output byte 8.Comment = ''; output byte 9.Name = 'output byte 9'; output byte 9.DataType = 'USINT'; output byte 9.Default = ''; output byte 9.Comment = ''; output byte 10.Name = 'output byte 10'; output byte 10.DataType = 'USINT'; output byte 10.Default = ''; output byte 10.Comment = ''; output byte 11.Name = 'output byte 11'; output byte 11.DataType = 'USINT'; output byte 11.Default = ''; output byte 11.Comment = ''; output byte 12.Name = 'output byte 12'; output byte 12.DataType = 'USINT'; output byte 12.Default = ''; output byte 12.Comment = ''; output byte 13.Name = 'output byte 13';
            output byte 13.DataType = 'USINT'; output byte 13.Default = ''; output byte 13.Comment = ''; output byte 14.Name = 'output byte 14'; output byte 14.DataType = 'USINT'; output byte 14.Default = ''; output byte 14.Comment = ''; output byte 15.Name = 'output byte 15'; output byte 15.DataType = 'USINT'; output byte 15.Default = ''; output byte 15.Comment = ''; output byte 16.Name = 'output byte 16'; output byte 16.DataType = 'USINT'; output byte 16.Default = ''; output byte 16.Comment = ''; output byte 17.Name = 'output byte 17'; output byte 17.DataType = 'USINT'; output byte 17.Default = ''; output byte 17.Comment = ''; output byte 18.Name = 'output byte 18'; output byte 18.DataType = 'USINT'; output byte 18.Default = ''; output byte 18.Comment = ''; output byte 19.Name = 'output byte 19'; output byte 19.DataType = 'USINT'; output byte 19.Default = ''; output byte 19.Comment = ''; output byte 20.Name = 'output byte 20'; output byte 20.DataType = 'USINT'; output byte 20.Default = ''; output byte 20.Comment = ''; output byte 21.Name = 'output byte 21'; output byte 21.DataType = 'USINT'; output byte 21.Default = ''; output byte 21.Comment = ''; output byte 22.Name = 'output byte 22'; output byte 22.DataType = 'USINT'; output byte 22.Default = ''; output byte 22.Comment = ''; output byte 23.Name = 'output byte 23';
            output byte 23.DataType = 'USINT'; output byte 23.Default = ''; output byte 23.Comment = ''; output byte 24.Name = 'output byte 24'; output byte 24.DataType = 'USINT'; output byte 24.Default = ''; output byte 24.Comment = ''; output byte 25.Name = 'output byte 25'; output byte 25.DataType = 'USINT'; output byte 25.Default = ''; output byte 25.Comment = ''; output byte 26.Name = 'output byte 26'; output byte 26.DataType = 'USINT'; output byte 26.Default = ''; output byte 26.Comment = ''; output byte 27.Name = 'output byte 27'; output byte 27.DataType = 'USINT'; output byte 27.Default = ''; output byte 27.Comment = ''; output byte 28.Name = 'output byte 28'; output byte 28.DataType = 'USINT'; output byte 28.Default = ''; output byte 28.Comment = ''; output byte 29.Name = 'output byte 29'; output byte 29.DataType = 'USINT'; output byte 29.Default = ''; output byte 29.Comment = ''; output byte 30.Name = 'output byte 30'; output byte 30.DataType = 'USINT'; output byte 30.Default = ''; output byte 30.Comment = ''; output byte 31.Name = 'output byte 31'; output byte 31.DataType = 'USINT'; output byte 31.Default = ''; output byte 31.Comment = ''; PD (I/Q Pin2 + C/Q Pin4).Name = 'PD (I/Q Pin2 + C/Q Pin4)'; PD (I/Q Pin2 + C/Q Pin4).DataType = 'UINT'; PD (I/Q Pin2 + C/Q Pin4).Default = ''; PD (I/Q Pin2 + C/Q Pin4).Comment = ''; New Message Available Flag.Name = 'New Message Available Flag';
            New Message Available Flag.DataType = 'BIT'; New Message Available Flag.Default = ''; New Message Available Flag.Comment = ''; Dummy.Name = 'Dummy'; Dummy.DataType = ''; Dummy.Default = ''; Dummy.Comment = ''; State of IO-Link Port X01.Name = 'State of IO-Link Port X01'; State of IO-Link Port X01.DataType = 'USINT'; State of IO-Link Port X01.Default = ''; State of IO-Link Port X01.Comment = ''; State of IO-Link Port X02.Name = 'State of IO-Link Port X02'; State of IO-Link Port X02.DataType = 'USINT'; State of IO-Link Port X02.Default = ''; State of IO-Link Port X02.Comment = ''; State of IO-Link Port X03.Name = 'State of IO-Link Port X03'; State of IO-Link Port X03.DataType = 'USINT'; State of IO-Link Port X03.Default = ''; State of IO-Link Port X03.Comment = ''; State of IO-Link Port X04.Name = 'State of IO-Link Port X04'; State of IO-Link Port X04.DataType = 'USINT'; State of IO-Link Port X04.Default = ''; State of IO-Link Port X04.Comment = ''; State of IO-Link Port X05.Name = 'State of IO-Link Port X05'; State of IO-Link Port X05.DataType = 'USINT'; State of IO-Link Port X05.Default = ''; State of IO-Link Port X05.Comment = ''; State of IO-Link Port X06.Name = 'State of IO-Link Port X06'; State of IO-Link Port X06.DataType = 'USINT'; State of IO-Link Port X06.Default = ''; State of IO-Link Port X06.Comment = ''; State of IO-Link Port X07.Name = 'State of IO-Link Port X07'; State of IO-Link Port X07.DataType = 'USINT'; State of IO-Link Port X07.Default = ''; State of IO-Link Port X07.Comment = ''; State of IO-Link Port X08.Name = 'State of IO-Link Port X08'; State of IO-Link Port X08.DataType = 'USINT'; State of IO-Link Port X08.Default = ''; State of IO-Link Port X08.Comment = ''; input byte 0.Name = 'input byte 0';
            input byte 0.DataType = 'USINT'; input byte 0.Default = ''; input byte 0.Comment = ''; input byte 1.Name = 'input byte 1'; input byte 1.DataType = 'USINT'; input byte 1.Default = ''; input byte 1.Comment = ''; input byte 2.Name = 'input byte 2'; input byte 2.DataType = 'USINT'; input byte 2.Default = ''; input byte 2.Comment = ''; input byte 3.Name = 'input byte 3'; input byte 3.DataType = 'USINT'; input byte 3.Default = ''; input byte 3.Comment = ''; input byte 4.Name = 'input byte 4'; input byte 4.DataType = 'USINT'; input byte 4.Default = ''; input byte 4.Comment = ''; input byte 5.Name = 'input byte 5'; input byte 5.DataType = 'USINT'; input byte 5.Default = ''; input byte 5.Comment = ''; input byte 6.Name = 'input byte 6'; input byte 6.DataType = 'USINT'; input byte 6.Default = ''; input byte 6.Comment = ''; input byte 7.Name = 'input byte 7'; input byte 7.DataType = 'USINT'; input byte 7.Default = ''; input byte 7.Comment = ''; input byte 0.Name = 'input byte 0'; input byte 0.DataType = 'USINT'; input byte 0.Default = ''; input byte 0.Comment = ''; input byte 1.Name = 'input byte 1'; input byte 1.DataType = 'USINT'; input byte 1.Default = ''; input byte 1.Comment = ''; input byte 0.Name = 'input byte 0';
            input byte 0.DataType = 'USINT'; input byte 0.Default = ''; input byte 0.Comment = ''; input byte 1.Name = 'input byte 1'; input byte 1.DataType = 'USINT'; input byte 1.Default = ''; input byte 1.Comment = ''; PD (C/Q Pin4).Name = 'PD (C/Q Pin4)'; PD (C/Q Pin4).DataType = 'USINT'; PD (C/Q Pin4).Default = ''; PD (C/Q Pin4).Comment = ''; input byte 0.Name = 'input byte 0'; input byte 0.DataType = 'USINT'; input byte 0.Default = ''; input byte 0.Comment = ''; input byte 1.Name = 'input byte 1'; input byte 1.DataType = 'USINT'; input byte 1.Default = ''; input byte 1.Comment = ''; input byte 2.Name = 'input byte 2'; input byte 2.DataType = 'USINT'; input byte 2.Default = ''; input byte 2.Comment = ''; input byte 3.Name = 'input byte 3'; input byte 3.DataType = 'USINT'; input byte 3.Default = ''; input byte 3.Comment = ''; input byte 4.Name = 'input byte 4'; input byte 4.DataType = 'USINT'; input byte 4.Default = ''; input byte 4.Comment = ''; input byte 5.Name = 'input byte 5'; input byte 5.DataType = 'USINT'; input byte 5.Default = ''; input byte 5.Comment = ''; input byte 6.Name = 'input byte 6'; input byte 6.DataType = 'USINT'; input byte 6.Default = ''; input byte 6.Comment = ''; input byte 7.Name = 'input byte 7';
            input byte 7.DataType = 'USINT'; input byte 7.Default = ''; input byte 7.Comment = ''; input byte 8.Name = 'input byte 8'; input byte 8.DataType = 'USINT'; input byte 8.Default = ''; input byte 8.Comment = ''; input byte 9.Name = 'input byte 9'; input byte 9.DataType = 'USINT'; input byte 9.Default = ''; input byte 9.Comment = ''; input byte 10.Name = 'input byte 10'; input byte 10.DataType = 'USINT'; input byte 10.Default = ''; input byte 10.Comment = ''; input byte 11.Name = 'input byte 11'; input byte 11.DataType = 'USINT'; input byte 11.Default = ''; input byte 11.Comment = ''; input byte 12.Name = 'input byte 12'; input byte 12.DataType = 'USINT'; input byte 12.Default = ''; input byte 12.Comment = ''; input byte 13.Name = 'input byte 13'; input byte 13.DataType = 'USINT'; input byte 13.Default = ''; input byte 13.Comment = ''; input byte 14.Name = 'input byte 14'; input byte 14.DataType = 'USINT'; input byte 14.Default = ''; input byte 14.Comment = ''; input byte 15.Name = 'input byte 15'; input byte 15.DataType = 'USINT'; input byte 15.Default = ''; input byte 15.Comment = ''; input byte 16.Name = 'input byte 16'; input byte 16.DataType = 'USINT'; input byte 16.Default = ''; input byte 16.Comment = ''; input byte 17.Name = 'input byte 17';
            input byte 17.DataType = 'USINT'; input byte 17.Default = ''; input byte 17.Comment = ''; input byte 18.Name = 'input byte 18'; input byte 18.DataType = 'USINT'; input byte 18.Default = ''; input byte 18.Comment = ''; input byte 19.Name = 'input byte 19'; input byte 19.DataType = 'USINT'; input byte 19.Default = ''; input byte 19.Comment = ''; input byte 20.Name = 'input byte 20'; input byte 20.DataType = 'USINT'; input byte 20.Default = ''; input byte 20.Comment = ''; input byte 21.Name = 'input byte 21'; input byte 21.DataType = 'USINT'; input byte 21.Default = ''; input byte 21.Comment = ''; input byte 22.Name = 'input byte 22'; input byte 22.DataType = 'USINT'; input byte 22.Default = ''; input byte 22.Comment = ''; input byte 23.Name = 'input byte 23'; input byte 23.DataType = 'USINT'; input byte 23.Default = ''; input byte 23.Comment = ''; input byte 24.Name = 'input byte 24'; input byte 24.DataType = 'USINT'; input byte 24.Default = ''; input byte 24.Comment = ''; input byte 25.Name = 'input byte 25'; input byte 25.DataType = 'USINT'; input byte 25.Default = ''; input byte 25.Comment = ''; input byte 26.Name = 'input byte 26'; input byte 26.DataType = 'USINT'; input byte 26.Default = ''; input byte 26.Comment = ''; input byte 27.Name = 'input byte 27';
            input byte 27.DataType = 'USINT'; input byte 27.Default = ''; input byte 27.Comment = ''; input byte 28.Name = 'input byte 28'; input byte 28.DataType = 'USINT'; input byte 28.Default = ''; input byte 28.Comment = ''; input byte 29.Name = 'input byte 29'; input byte 29.DataType = 'USINT'; input byte 29.Default = ''; input byte 29.Comment = ''; input byte 30.Name = 'input byte 30'; input byte 30.DataType = 'USINT'; input byte 30.Default = ''; input byte 30.Comment = ''; input byte 31.Name = 'input byte 31'; input byte 31.DataType = 'USINT'; input byte 31.Default = ''; input byte 31.Comment = ''; PD (C/Q Pin4).Name = 'PD (C/Q Pin4)'; PD (C/Q Pin4).DataType = 'USINT'; PD (C/Q Pin4).Default = ''; PD (C/Q Pin4).Comment = ''
          output Application.GVL_IO.xIOFLD_02_X02_P2_Out : BOOL  // PD (I/Q Pin2).Bit1
          output Application.GVL_IO.xIOFLD_02_X04_P2_Out : BOOL  // PD (I/Q Pin2).Bit3
          input  Application.GVL_IO.xIOFLD_02_X06_P2_In : BOOL  // PD (I/Q Pin2 + C/Q Pin4).Bit5
          input  Application.GVL_IO.xIOFLD_02_X08_P2_In : BOOL  // PD (I/Q Pin2 + C/Q Pin4).Bit7
          unmapped channels: PD (I/Q Pin2), PD (I/Q Pin2 + C/Q Pin4), New Message Available Flag, Dummy, Dummy, Dummy, Dummy, Dummy, Dummy, Dummy, State of IO-Link Port X01, State of IO-Link Port X02, State of IO-Link Port X03, State of IO-Link Port X04, State of IO-Link Port X05, State of IO-Link Port X06, State of IO-Link Port X07, State of IO-Link Port X08
        IO_Link_Port_X01 : IO-Link 8 Byte Input / 8 Byte Output Process Data , WAGO Kontakttechnik GmbH u. Co. KG, order no. IOL_8/8_I/O-Bytes, version 0
            settings: Number of Outputs = 8; Number of Inputs = 8; Number of Infos about Outputs = 8; Number of Infos about Inputs = 8; RxTxPdo.Fixed = False; RxTxPdo.Mandatory = False; RxTxPdo.Virtual = False; RxTxPdo.DependOnSlot = True; RxTxPdo.DependOnSlotGroup = False; RxTxPdo.OverwrittenByModule = True; output byte 0.Offset = 0; output byte 0.DependOnSlot = True; output byte 0.DependOnSlotGroup = False; output byte 1.Offset = 0; output byte 1.DependOnSlot = True; output byte 1.DependOnSlotGroup = False; output byte 2.Offset = 0; output byte 2.DependOnSlot = True; output byte 2.DependOnSlotGroup = False; output byte 3.Offset = 0; output byte 3.DependOnSlot = True; output byte 3.DependOnSlotGroup = False; output byte 4.Offset = 0; output byte 4.DependOnSlot = True; output byte 4.DependOnSlotGroup = False; output byte 5.Offset = 0; output byte 5.DependOnSlot = True; output byte 5.DependOnSlotGroup = False; output byte 6.Offset = 0; output byte 6.DependOnSlot = True; output byte 6.DependOnSlotGroup = False; output byte 7.Offset = 0; output byte 7.DependOnSlot = True; output byte 7.DependOnSlotGroup = False; RxTxPdo.Fixed = False; RxTxPdo.Mandatory = False; RxTxPdo.Virtual = False; RxTxPdo.DependOnSlot = True; RxTxPdo.DependOnSlotGroup = False; RxTxPdo.OverwrittenByModule = True;
              input byte 0.Offset = 0; input byte 0.DependOnSlot = True; input byte 0.DependOnSlotGroup = False; input byte 1.Offset = 0; input byte 1.DependOnSlot = True; input byte 1.DependOnSlotGroup = False; input byte 2.Offset = 0; input byte 2.DependOnSlot = True; input byte 2.DependOnSlotGroup = False; input byte 3.Offset = 0; input byte 3.DependOnSlot = True; input byte 3.DependOnSlotGroup = False; input byte 4.Offset = 0; input byte 4.DependOnSlot = True; input byte 4.DependOnSlotGroup = False; input byte 5.Offset = 0; input byte 5.DependOnSlot = True; input byte 5.DependOnSlotGroup = False; input byte 6.Offset = 0; input byte 6.DependOnSlot = True; input byte 6.DependOnSlotGroup = False; input byte 7.Offset = 0; input byte 7.DependOnSlot = True; input byte 7.DependOnSlotGroup = False; output byte 0.Default = ''; output byte 1.Default = ''; output byte 2.Default = ''; output byte 3.Default = ''; output byte 4.Default = ''; output byte 5.Default = ''; output byte 6.Default = ''; output byte 7.Default = ''; input byte 0.Default = ''; input byte 1.Default = ''; input byte 2.Default = ''; input byte 3.Default = ''; input byte 4.Default = ''; input byte 5.Default = ''; input byte 6.Default = ''; input byte 7.Default = ''
            unmapped channels: output byte 0, output byte 1, output byte 2, output byte 3, output byte 4, output byte 5, output byte 6, output byte 7, input byte 0, input byte 1, input byte 2, input byte 3, input byte 4, input byte 5, input byte 6, input byte 7
        IO_Link_Port_X02 : Digital Output, WAGO Kontakttechnik GmbH u. Co. KG, order no. Digital_OUT, version 0
            settings: Number of Outputs = 1; Number of Infos about Outputs = 1; RxTxPdo.Fixed = False; RxTxPdo.Mandatory = False; RxTxPdo.Virtual = False; RxTxPdo.DependOnSlot = True; RxTxPdo.DependOnSlotGroup = False; RxTxPdo.OverwrittenByModule = True; PD (C/Q Pin4).Offset = 0; PD (C/Q Pin4).DependOnSlot = True; PD (C/Q Pin4).DependOnSlotGroup = False; PD (C/Q Pin4).Default = ''
            output Application.GVL_IO.xIOFLD_02_X02_P4_Out : BOOL  // PD (C/Q Pin4).Bit0
            unmapped channels: PD (C/Q Pin4)
        IO_Link_Port_X03 : IO-Link 2 Byte Input / 2 Byte Output Process Data , WAGO Kontakttechnik GmbH u. Co. KG, order no. IOL_2/2_I/O-Bytes, version 0
            settings: Number of Outputs = 2; Number of Inputs = 2; Number of Infos about Outputs = 2; Number of Infos about Inputs = 2; RxTxPdo.Fixed = False; RxTxPdo.Mandatory = False; RxTxPdo.Virtual = False; RxTxPdo.DependOnSlot = True; RxTxPdo.DependOnSlotGroup = False; RxTxPdo.OverwrittenByModule = True; output byte 0.Offset = 0; output byte 0.DependOnSlot = True; output byte 0.DependOnSlotGroup = False; output byte 1.Offset = 0; output byte 1.DependOnSlot = True; output byte 1.DependOnSlotGroup = False; RxTxPdo.Fixed = False; RxTxPdo.Mandatory = False; RxTxPdo.Virtual = False; RxTxPdo.DependOnSlot = True; RxTxPdo.DependOnSlotGroup = False; RxTxPdo.OverwrittenByModule = True; input byte 0.Offset = 0; input byte 0.DependOnSlot = True; input byte 0.DependOnSlotGroup = False; input byte 1.Offset = 0; input byte 1.DependOnSlot = True; input byte 1.DependOnSlotGroup = False; output byte 0.Default = ''; output byte 1.Default = ''; input byte 0.Default = ''; input byte 1.Default = ''
            unmapped channels: output byte 0, output byte 1, input byte 0, input byte 1
        IO_Link_Port_X04 : Digital Output, WAGO Kontakttechnik GmbH u. Co. KG, order no. Digital_OUT, version 0
            settings: Number of Outputs = 1; Number of Infos about Outputs = 1; RxTxPdo.Fixed = False; RxTxPdo.Mandatory = False; RxTxPdo.Virtual = False; RxTxPdo.DependOnSlot = True; RxTxPdo.DependOnSlotGroup = False; RxTxPdo.OverwrittenByModule = True; PD (C/Q Pin4).Offset = 0; PD (C/Q Pin4).DependOnSlot = True; PD (C/Q Pin4).DependOnSlotGroup = False; PD (C/Q Pin4).Default = ''
            output Application.GVL_IO.xIOFLD_02_X04_P4_Out : BOOL  // PD (C/Q Pin4).Bit0
            output Application.GVL_IO.xIOFLD_02_X04_P2_Out : BOOL  // PD (C/Q Pin4).Bit1
            unmapped channels: PD (C/Q Pin4)
        IO_Link_Port_X05 : IO-Link 2 Byte Input / 2 Byte Output Process Data , WAGO Kontakttechnik GmbH u. Co. KG, order no. IOL_2/2_I/O-Bytes, version 0
            settings: Number of Outputs = 2; Number of Inputs = 2; Number of Infos about Outputs = 2; Number of Infos about Inputs = 2; RxTxPdo.Fixed = False; RxTxPdo.Mandatory = False; RxTxPdo.Virtual = False; RxTxPdo.DependOnSlot = True; RxTxPdo.DependOnSlotGroup = False; RxTxPdo.OverwrittenByModule = True; output byte 0.Offset = 0; output byte 0.DependOnSlot = True; output byte 0.DependOnSlotGroup = False; output byte 1.Offset = 0; output byte 1.DependOnSlot = True; output byte 1.DependOnSlotGroup = False; RxTxPdo.Fixed = False; RxTxPdo.Mandatory = False; RxTxPdo.Virtual = False; RxTxPdo.DependOnSlot = True; RxTxPdo.DependOnSlotGroup = False; RxTxPdo.OverwrittenByModule = True; input byte 0.Offset = 0; input byte 0.DependOnSlot = True; input byte 0.DependOnSlotGroup = False; input byte 1.Offset = 0; input byte 1.DependOnSlot = True; input byte 1.DependOnSlotGroup = False; output byte 0.Default = ''; output byte 1.Default = ''; input byte 0.Default = ''; input byte 1.Default = ''
            unmapped channels: output byte 0, output byte 1, input byte 0, input byte 1
        IO_Link_Port_X06 : Digital Input, WAGO Kontakttechnik GmbH u. Co. KG, order no. Digital_IN, version 0
            settings: Number of Inputs = 1; Number of Infos about Inputs = 1; RxTxPdo.Fixed = False; RxTxPdo.Mandatory = False; RxTxPdo.Virtual = False; RxTxPdo.DependOnSlot = True; RxTxPdo.DependOnSlotGroup = False; RxTxPdo.OverwrittenByModule = True; PD (C/Q Pin4).Offset = 0; PD (C/Q Pin4).DependOnSlot = True; PD (C/Q Pin4).DependOnSlotGroup = False; PD (C/Q Pin4).Default = ''
            unmapped channels: PD (C/Q Pin4)
        IO_Link_Port_X07 : IO-Link 32 Byte Input / 32 Byte Output Process Data, WAGO Kontakttechnik GmbH u. Co. KG, order no. IOL_32/32_I/O-Bytes, version 0
            settings: Number of Outputs = 32; Number of Inputs = 32; Number of Infos about Outputs = 32; Number of Infos about Inputs = 32; RxTxPdo.Fixed = False; RxTxPdo.Mandatory = False; RxTxPdo.Virtual = False; RxTxPdo.DependOnSlot = True; RxTxPdo.DependOnSlotGroup = False; RxTxPdo.OverwrittenByModule = True; output byte 0.Offset = 0; output byte 0.DependOnSlot = True; output byte 0.DependOnSlotGroup = False; output byte 1.Offset = 0; output byte 1.DependOnSlot = True; output byte 1.DependOnSlotGroup = False; output byte 2.Offset = 0; output byte 2.DependOnSlot = True; output byte 2.DependOnSlotGroup = False; output byte 3.Offset = 0; output byte 3.DependOnSlot = True; output byte 3.DependOnSlotGroup = False; output byte 4.Offset = 0; output byte 4.DependOnSlot = True; output byte 4.DependOnSlotGroup = False; output byte 5.Offset = 0; output byte 5.DependOnSlot = True; output byte 5.DependOnSlotGroup = False; output byte 6.Offset = 0; output byte 6.DependOnSlot = True; output byte 6.DependOnSlotGroup = False; output byte 7.Offset = 0; output byte 7.DependOnSlot = True; output byte 7.DependOnSlotGroup = False; output byte 8.Offset = 0; output byte 8.DependOnSlot = True; output byte 8.DependOnSlotGroup = False; output byte 9.Offset = 0; output byte 9.DependOnSlot = True; output byte 9.DependOnSlotGroup = False;
              output byte 10.Offset = 0; output byte 10.DependOnSlot = True; output byte 10.DependOnSlotGroup = False; output byte 11.Offset = 0; output byte 11.DependOnSlot = True; output byte 11.DependOnSlotGroup = False; output byte 12.Offset = 0; output byte 12.DependOnSlot = True; output byte 12.DependOnSlotGroup = False; output byte 13.Offset = 0; output byte 13.DependOnSlot = True; output byte 13.DependOnSlotGroup = False; output byte 14.Offset = 0; output byte 14.DependOnSlot = True; output byte 14.DependOnSlotGroup = False; output byte 15.Offset = 0; output byte 15.DependOnSlot = True; output byte 15.DependOnSlotGroup = False; output byte 16.Offset = 0; output byte 16.DependOnSlot = True; output byte 16.DependOnSlotGroup = False; output byte 17.Offset = 0; output byte 17.DependOnSlot = True; output byte 17.DependOnSlotGroup = False; output byte 18.Offset = 0; output byte 18.DependOnSlot = True; output byte 18.DependOnSlotGroup = False; output byte 19.Offset = 0; output byte 19.DependOnSlot = True; output byte 19.DependOnSlotGroup = False; output byte 20.Offset = 0; output byte 20.DependOnSlot = True; output byte 20.DependOnSlotGroup = False; output byte 21.Offset = 0; output byte 21.DependOnSlot = True; output byte 21.DependOnSlotGroup = False; output byte 22.Offset = 0; output byte 22.DependOnSlot = True; output byte 22.DependOnSlotGroup = False; output byte 23.Offset = 0;
              output byte 23.DependOnSlot = True; output byte 23.DependOnSlotGroup = False; output byte 24.Offset = 0; output byte 24.DependOnSlot = True; output byte 24.DependOnSlotGroup = False; output byte 25.Offset = 0; output byte 25.DependOnSlot = True; output byte 25.DependOnSlotGroup = False; output byte 26.Offset = 0; output byte 26.DependOnSlot = True; output byte 26.DependOnSlotGroup = False; output byte 27.Offset = 0; output byte 27.DependOnSlot = True; output byte 27.DependOnSlotGroup = False; output byte 28.Offset = 0; output byte 28.DependOnSlot = True; output byte 28.DependOnSlotGroup = False; output byte 29.Offset = 0; output byte 29.DependOnSlot = True; output byte 29.DependOnSlotGroup = False; output byte 30.Offset = 0; output byte 30.DependOnSlot = True; output byte 30.DependOnSlotGroup = False; output byte 31.Offset = 0; output byte 31.DependOnSlot = True; output byte 31.DependOnSlotGroup = False; RxTxPdo.Fixed = False; RxTxPdo.Mandatory = False; RxTxPdo.Virtual = False; RxTxPdo.DependOnSlot = True; RxTxPdo.DependOnSlotGroup = False; RxTxPdo.OverwrittenByModule = True; input byte 0.Offset = 0; input byte 0.DependOnSlot = True; input byte 0.DependOnSlotGroup = False; input byte 1.Offset = 0; input byte 1.DependOnSlot = True; input byte 1.DependOnSlotGroup = False; input byte 2.Offset = 0; input byte 2.DependOnSlot = True;
              input byte 2.DependOnSlotGroup = False; input byte 3.Offset = 0; input byte 3.DependOnSlot = True; input byte 3.DependOnSlotGroup = False; input byte 4.Offset = 0; input byte 4.DependOnSlot = True; input byte 4.DependOnSlotGroup = False; input byte 5.Offset = 0; input byte 5.DependOnSlot = True; input byte 5.DependOnSlotGroup = False; input byte 6.Offset = 0; input byte 6.DependOnSlot = True; input byte 6.DependOnSlotGroup = False; input byte 7.Offset = 0; input byte 7.DependOnSlot = True; input byte 7.DependOnSlotGroup = False; input byte 8.Offset = 0; input byte 8.DependOnSlot = True; input byte 8.DependOnSlotGroup = False; input byte 9.Offset = 0; input byte 9.DependOnSlot = True; input byte 9.DependOnSlotGroup = False; input byte 10.Offset = 0; input byte 10.DependOnSlot = True; input byte 10.DependOnSlotGroup = False; input byte 11.Offset = 0; input byte 11.DependOnSlot = True; input byte 11.DependOnSlotGroup = False; input byte 12.Offset = 0; input byte 12.DependOnSlot = True; input byte 12.DependOnSlotGroup = False; input byte 13.Offset = 0; input byte 13.DependOnSlot = True; input byte 13.DependOnSlotGroup = False; input byte 14.Offset = 0; input byte 14.DependOnSlot = True; input byte 14.DependOnSlotGroup = False; input byte 15.Offset = 0; input byte 15.DependOnSlot = True; input byte 15.DependOnSlotGroup = False;
              input byte 16.Offset = 0; input byte 16.DependOnSlot = True; input byte 16.DependOnSlotGroup = False; input byte 17.Offset = 0; input byte 17.DependOnSlot = True; input byte 17.DependOnSlotGroup = False; input byte 18.Offset = 0; input byte 18.DependOnSlot = True; input byte 18.DependOnSlotGroup = False; input byte 19.Offset = 0; input byte 19.DependOnSlot = True; input byte 19.DependOnSlotGroup = False; input byte 20.Offset = 0; input byte 20.DependOnSlot = True; input byte 20.DependOnSlotGroup = False; input byte 21.Offset = 0; input byte 21.DependOnSlot = True; input byte 21.DependOnSlotGroup = False; input byte 22.Offset = 0; input byte 22.DependOnSlot = True; input byte 22.DependOnSlotGroup = False; input byte 23.Offset = 0; input byte 23.DependOnSlot = True; input byte 23.DependOnSlotGroup = False; input byte 24.Offset = 0; input byte 24.DependOnSlot = True; input byte 24.DependOnSlotGroup = False; input byte 25.Offset = 0; input byte 25.DependOnSlot = True; input byte 25.DependOnSlotGroup = False; input byte 26.Offset = 0; input byte 26.DependOnSlot = True; input byte 26.DependOnSlotGroup = False; input byte 27.Offset = 0; input byte 27.DependOnSlot = True; input byte 27.DependOnSlotGroup = False; input byte 28.Offset = 0; input byte 28.DependOnSlot = True; input byte 28.DependOnSlotGroup = False; input byte 29.Offset = 0;
              input byte 29.DependOnSlot = True; input byte 29.DependOnSlotGroup = False; input byte 30.Offset = 0; input byte 30.DependOnSlot = True; input byte 30.DependOnSlotGroup = False; input byte 31.Offset = 0; input byte 31.DependOnSlot = True; input byte 31.DependOnSlotGroup = False; output byte 0.Default = ''; output byte 1.Default = ''; output byte 2.Default = ''; output byte 3.Default = ''; output byte 4.Default = ''; output byte 5.Default = ''; output byte 6.Default = ''; output byte 7.Default = ''; output byte 8.Default = ''; output byte 9.Default = ''; output byte 10.Default = ''; output byte 11.Default = ''; output byte 12.Default = ''; output byte 13.Default = ''; output byte 14.Default = ''; output byte 15.Default = ''; output byte 16.Default = ''; output byte 17.Default = ''; output byte 18.Default = ''; output byte 19.Default = ''; output byte 20.Default = ''; output byte 21.Default = ''; output byte 22.Default = ''; output byte 23.Default = ''; output byte 24.Default = ''; output byte 25.Default = ''; output byte 26.Default = ''; output byte 27.Default = ''; output byte 28.Default = ''; output byte 29.Default = ''; output byte 30.Default = ''; output byte 31.Default = '';
              input byte 0.Default = ''; input byte 1.Default = ''; input byte 2.Default = ''; input byte 3.Default = ''; input byte 4.Default = ''; input byte 5.Default = ''; input byte 6.Default = ''; input byte 7.Default = ''; input byte 8.Default = ''; input byte 9.Default = ''; input byte 10.Default = ''; input byte 11.Default = ''; input byte 12.Default = ''; input byte 13.Default = ''; input byte 14.Default = ''; input byte 15.Default = ''; input byte 16.Default = ''; input byte 17.Default = ''; input byte 18.Default = ''; input byte 19.Default = ''; input byte 20.Default = ''; input byte 21.Default = ''; input byte 22.Default = ''; input byte 23.Default = ''; input byte 24.Default = ''; input byte 25.Default = ''; input byte 26.Default = ''; input byte 27.Default = ''; input byte 28.Default = ''; input byte 29.Default = ''; input byte 30.Default = ''; input byte 31.Default = ''
            unmapped channels: output byte 0, output byte 1, output byte 2, output byte 3, output byte 4, output byte 5, output byte 6, output byte 7, output byte 8, output byte 9, output byte 10, output byte 11, output byte 12, output byte 13, output byte 14, output byte 15, output byte 16, output byte 17, output byte 18, output byte 19, output byte 20, output byte 21, output byte 22, output byte 23, output byte 24, output byte 25, output byte 26, output byte 27, output byte 28, output byte 29, output byte 30, output byte 31, input byte 0, input byte 1, input byte 2, input byte 3, input byte 4, input byte 5, input byte 6, input byte 7,
              input byte 8, input byte 9, input byte 10, input byte 11, input byte 12, input byte 13, input byte 14, input byte 15, input byte 16, input byte 17, input byte 18, input byte 19, input byte 20, input byte 21, input byte 22, input byte 23, input byte 24, input byte 25, input byte 26, input byte 27, input byte 28, input byte 29, input byte 30, input byte 31
        IO_Link_Port_X08 : Digital Input, WAGO Kontakttechnik GmbH u. Co. KG, order no. Digital_IN, version 0
            settings: Number of Inputs = 1; Number of Infos about Inputs = 1; RxTxPdo.Fixed = False; RxTxPdo.Mandatory = False; RxTxPdo.Virtual = False; RxTxPdo.DependOnSlot = True; RxTxPdo.DependOnSlotGroup = False; RxTxPdo.OverwrittenByModule = True; PD (C/Q Pin4).Offset = 0; PD (C/Q Pin4).DependOnSlot = True; PD (C/Q Pin4).DependOnSlotGroup = False; PD (C/Q Pin4).Default = ''
            unmapped channels: PD (C/Q Pin4)
    Kbus : Kbus, WAGO, version 2.1.0.1
        unmapped channels: K-BUS diagnostics
      _750_1657_24 : 750-1657#24, WAGO, order no. 750-1657, version 2.0.0.15
          unmapped channels: _INPUTCHANNEL, _OUTPUTCHANNEL
      _75x_4DI : 75x-4DI, WAGO, version 2.0.0.13
          unmapped channels: _IN
      _75x_4DO : 75x-4DO, WAGO, version 2.0.0.13
          output Application.PLC_PRG.xWD : BOOL  // _OUT._OUT
          output Application.PLC_PRG.xWD_ : BOOL  // _OUT._OUT
          unmapped channels: _OUT
    Serial
      COM1 : COM1, WAGO, version 0.0.0.19
*)

// Device/Application/GVL_IO
{attribute 'qualified_only'}
VAR_GLOBAL
	xIOFLD_01_X01_P2_In				: BOOL;
	xIOFLD_01_X01_P4_In				: BOOL;
	xIOFLD_01_X02_P2_Out			: BOOL;
	xIOFLD_01_X02_P4_Out			: BOOL;
	xIOFLD_01_X03_P2_In				: BOOL;
	xIOFLD_01_X03_P4_In				: BOOL;
	xIOFLD_01_X04_P2_Out			: BOOL;
	xIOFLD_01_X04_P4_Out			: BOOL;
	xIOFLD_01_X05_P2_In				: BOOL;
	xIOFLD_01_X05_P4_In				: BOOL;
	xIOFLD_01_X06_P2_Out			: BOOL;
	xIOFLD_01_X06_P4_Out			: BOOL;
	xIOFLD_01_X07_P2_In				: BOOL;
	xIOFLD_01_X07_P4_In				: BOOL;
	xIOFLD_01_X08_P2_Out			: BOOL;
	xIOFLD_01_X08_P4_Out			: BOOL;	
	
	xIOFLD_02_X02_P2_Out			: BOOL;
	xIOFLD_02_X02_P4_Out			: BOOL;
	xIOFLD_02_X04_P2_Out			: BOOL;
	xIOFLD_02_X04_P4_Out			: BOOL;
	xIOFLD_02_X06_P2_In				: BOOL;
	xIOFLD_02_X06_P4_In				: BOOL;
	xIOFLD_02_X08_P2_In				: BOOL;
	xIOFLD_02_X08_P4_In				: BOOL;
END_VAR

// Device/Application/PLC_PRG
PROGRAM PLC_PRG
VAR
	uiCnt				: UINT;
	xWD					: BOOL;
	xWD_				: BOOL;
	
END_VAR

(* PLC cycle counter and watchdog *)
uiCnt := uiCnt + 1;
xWD := uiCnt.3;
xWD_ := NOT xWD;

(* read-write 765-1202 IO's *)
GVL_IO.xIOFLD_01_X01_P2_In;
GVL_IO.xIOFLD_01_X01_P4_In;
GVL_IO.xIOFLD_01_X02_P2_Out	:= xWD;
GVL_IO.xIOFLD_01_X02_P4_Out := xWD_;
GVL_IO.xIOFLD_01_X03_P2_In;
GVL_IO.xIOFLD_01_X03_P4_In;
GVL_IO.xIOFLD_01_X04_P2_Out	:= xWD;
GVL_IO.xIOFLD_01_X04_P4_Out := xWD_;
GVL_IO.xIOFLD_01_X05_P2_In;
GVL_IO.xIOFLD_01_X05_P4_In;
GVL_IO.xIOFLD_01_X06_P2_Out	:= xWD;
GVL_IO.xIOFLD_01_X06_P4_Out := xWD_;
GVL_IO.xIOFLD_01_X07_P2_In;
GVL_IO.xIOFLD_01_X07_P4_In;
GVL_IO.xIOFLD_01_X08_P2_Out	:= xWD;
GVL_IO.xIOFLD_01_X08_P4_Out := xWD_;

(* read-write 765-4201 IO's *)
GVL_IO.xIOFLD_02_X02_P2_Out := xWD;
GVL_IO.xIOFLD_02_X02_P4_Out := xWD_;
GVL_IO.xIOFLD_02_X04_P2_Out := xWD;
GVL_IO.xIOFLD_02_X04_P4_Out := xWD_;
GVL_IO.xIOFLD_02_X06_P2_In;
GVL_IO.xIOFLD_02_X06_P4_In;
GVL_IO.xIOFLD_02_X08_P2_In;
GVL_IO.xIOFLD_02_X08_P4_In;

(* IOL-call *)
PRG_IOL_Call();

END_PROGRAM

// Device/Application/PRG_IOL_Call
PROGRAM PRG_IOL_Call
VAR
	usiIOL_Call_Com				: USINT := 1;
	usiIOL_Call_Channel			: USINT;
	udiIOL_Call_Timeout			: UDINT := 300;
	usiIOL_Call_Port			: USINT := 1;
	uiIOL_Call_Index			: UINT := 0;
	usiIOL_Call_SubIndex		: USINT := 0;
	udiIOL_Call_ReadWriteLen	: UDINT;
	aIOL_Call_Data				: ARRAY[0..9] OF BYTE;
	
	
		
	oIOL_Call_Read				: ETC_ADS_IoLinkRead;
	xIOL_Call_Read_Execute		: BOOL;
	xIOL_Call_Read_Abort		: BOOL;
	xIOL_Call_Read_Done			: BOOL;
	xIOL_Call_Read_Busy			: BOOL;
	xIOL_Call_Read_Err			: BOOL;
	xIOL_Call_Read_Aborted		: BOOL;
	udiIOL_Call_Read_RespErr	: UDINT;
	udiIOL_Call_Read_DataRD		: UDINT;
		
	oIOL_Call_Write				: ETC_ADS_IoLinkWrite;
	xIOL_Call_Write_Execute		: BOOL;
	xIOL_Call_Write_Abort		: BOOL;
	xIOL_Call_Write_Done		: BOOL;
	xIOL_Call_Write_Busy		: BOOL;
	xIOL_Call_Write_Err			: BOOL;
	xIOL_Call_Write_Aborted		: BOOL;
	udiIOL_Call_Write_RespErr	: UDINT;
	udiIOL_Call_Write_DataWR	: UDINT;
END_VAR
VAR CONSTANT
	c_udiIndexGroup				: UDINT := 16#F302;
END_VAR


(* call instances *)
oIOL_Call_Read(
	xExecute:= xIOL_Call_Read_Execute, 
	xAbort:= xIOL_Call_Read_Abort, 
	xDone=> xIOL_Call_Read_Done, 
	xBusy=> xIOL_Call_Read_Busy, 
	xError=> xIOL_Call_Read_Err, 
	xAborted=> xIOL_Call_Read_Aborted, 
	usiCom:= usiIOL_Call_Com, 
	uiDevice:= IOFLD_02_765_4201.PhysSlaveAddr, 
	usiChannel:= usiIOL_Call_Channel, 
	udiTimeout:= udiIOL_Call_Timeout, 
	usiPort:= usiIOL_Call_Port, 
	uiIndex:= uiIOL_Call_Index, 
	usiSubIndex:= usiIOL_Call_SubIndex, 
	udiSize:= udiIOL_Call_ReadWriteLen, 
	pbyData:= ADR(aIOL_Call_Data), 
	udiIndexGroup:= c_udiIndexGroup, 
	udiResponseError=> udiIOL_Call_Read_RespErr, 
	udiDataRead=> udiIOL_Call_Read_DataRD);
	
oIOL_Call_Write(
	xExecute:= xIOL_Call_Write_Execute, 
	xAbort:= xIOL_Call_Write_Abort, 
	xDone=> xIOL_Call_Write_Done, 
	xBusy=> xIOL_Call_Write_Busy, 
	xError=> xIOL_Call_Write_Err, 
	xAborted=> xIOL_Call_Write_Aborted, 
	usiCom:= usiIOL_Call_Com, 
	uiDevice:= IOFLD_02_765_4201.PhysSlaveAddr, 
	usiChannel:= usiIOL_Call_Channel, 
	udiTimeout:= udiIOL_Call_Timeout, 
	usiPort:= usiIOL_Call_Port, 
	uiIndex:= uiIOL_Call_Index, 
	usiSubIndex:= usiIOL_Call_SubIndex, 
	udiSize:= udiIOL_Call_ReadWriteLen, 
	pbyData:= ADR(aIOL_Call_Data), 
	udiIndexGroup:= c_udiIndexGroup, 
	udiResponseError=> udiIOL_Call_Write_RespErr, 
	udiDataWritten=> udiIOL_Call_Write_DataWR);

END_PROGRAM
